KUKA KRL program: EPS_2_251825_SA28_A_20260116064107.src

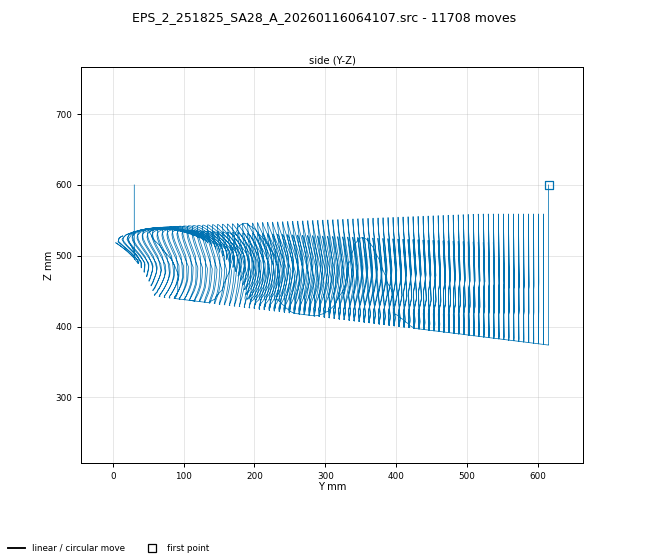
[picture p0: tool path of EPS_2_251825_SA28_A_20260116064107.src, 11708 of 11710 moves have a stored position in this frame; points joined in program order, loops and branches not executed]
&ACCESS RVP
&REL 4
&COMMENT QRS 19112012
&PARAM EDITMASK = *
DEF PART()
EXT BAS (BAS_COMMAND :IN,REAL :IN )
INT I
BAS (#INITMOV,0 )

;KUKA QRS Post kuka4.cps  Date:22-06-2017 !

File_ID=2987

QRS_PRE_INIT()

;Init var - Until changes are made in qrs_pre_init
Outlet_Square_prg=0
Inlet_1_Square_prg=0
Inlet_2_Square_prg=0
Inlet_3_Square_prg=0
Inlet_4_Square_prg=0
Inlet_5_Square_prg=0

Outlet_1={X 0.000, Y 520.860, Z 458.500, B 0.000, E1 0.000 }
Inlet_1={X 0.000, Y 523.760, Z 418.500, B 0.000, E1 223.000 }
Outlet_1_type=201
Inlet_1_type=201
;QRS#1=Sidecore dimensions
;QRS#2=200-8" PVC SDR 35
;QRS#3=200-8" PVC SDR 35
;QRS#4=
;QRS#5=
;QRS#6=
;QRS#7=
;QRS#8=
;QRS#9=12-08 PSX
;QRS#10=12-08 PSX
;QRS#11=
;QRS#12=
;QRS#13=
;QRS#14=
;QRS#15=
;QRS#16=1220x127x838 2,75'
;QRS#17=EPS Height
;QRS#18=559
;QRS#19=*
;QRS#20= UPDATED VERSION 22-06-2017
;QRS#21=*
Outlet_Square=0100
Inlet_1_Square=0100
Inlet_2_Square=0
Inlet_3_Square=0
Inlet_4_Square=0
Inlet_5_Square=0
Mill_Square=1
Outlet_Square_Prg=204
Inlet_1_Square_prg=204

QRS_INIT()

$ADVANCE=5

; T1
PTP {E1 173.612,E2 173.612}
PTP {X 0,Y 615.494,A -85,B 0,C 180,E1 173.612,E2 173.612,E3 0,E4 0,E5 0,E6 0}
QRS_SPEED_INIT()
LIN {X 0,Y 615.494,Z 600,A -85,B 0,C 180,E1 173.612,E2 173.612,E3 0,E4 0,E5 0,E6 0} C_VEL
LIN {X 0,Y 615.494,Z 383.874,A -85,B 0,C 180,E1 173.612,E2 173.612} C_VEL
LIN {X 0,Y 615.494,Z 375.697,A -85,B 0,C 180,E1 173.612,E2 173.612} C_VEL
LIN {X 0,Y 615.482,Z 373.697,A -85,B 0,C 180,E1 173.425,E2 173.425} C_VEL
LIN {X 0,Y 615.489,Z 373.696,A -85,B 0,C 180,E1 170.801,E2 170.801} C_VEL
LIN {X 0,Y 615.487,Z 373.7,A -85,B 0,C 180,E1 168.139,E2 168.139} C_VEL
LIN {X 0,Y 615.495,Z 373.697,A -85,B 0,C 180,E1 165.451,E2 165.451} C_VEL
LIN {X 0,Y 615.472,Z 373.699,A -85,B 0,C 180,E1 162.729,E2 162.729} C_VEL
LIN {X 0,Y 615.476,Z 373.7,A -85,B 0,C 180,E1 159.967,E2 159.967} C_VEL
LIN {X 0,Y 615.49,Z 373.699,A -85,B 0,C 180,E1 157.156,E2 157.156} C_VEL
LIN {X 0,Y 615.465,Z 373.701,A -85,B 0,C 180,E1 154.435,E2 154.435} C_VEL
LIN {X 0,Y 615.469,Z 373.7,A -85,B 0,C 180,E1 152.084,E2 152.084} C_VEL
LIN {X 0,Y 615.486,Z 373.698,A -85,B 0,C 180,E1 149.84,E2 149.84} C_VEL
LIN {X 0,Y 615.497,Z 373.697,A -85,B 0,C 180,E1 147.543,E2 147.543} C_VEL
LIN {X 0,Y 615.484,Z 373.7,A -85,B 0,C 180,E1 145.185,E2 145.185} C_VEL
LIN {X 0,Y 615.48,Z 373.7,A -85,B 0,C 180,E1 142.757,E2 142.757} C_VEL
LIN {X 0,Y 615.471,Z 373.699,A -85,B 0,C 180,E1 139.913,E2 139.913} C_VEL
LIN {X 0,Y 615.489,Z 373.701,A -85,B 0,C 180,E1 136.952,E2 136.952} C_VEL
LIN {X 0,Y 615.472,Z 373.699,A -85,B 0,C 180,E1 134.151,E2 134.151} C_VEL
LIN {X 0,Y 615.495,Z 373.694,A -85,B 0,C 180,E1 131.473,E2 131.473} C_VEL
LIN {X 0,Y 615.481,Z 373.7,A -85,B 0,C 180,E1 128.905,E2 128.905} C_VEL
LIN {X 0,Y 615.486,Z 373.7,A -85,B 0,C 180,E1 126.425,E2 126.425} C_VEL
LIN {X 0,Y 615.492,Z 373.696,A -85,B 0,C 180,E1 123.535,E2 123.535} C_VEL
LIN {X 0,Y 615.467,Z 373.7,A -85,B 0,C 180,E1 120.921,E2 120.921} C_VEL
LIN {X 0,Y 615.467,Z 373.7,A -85,B 0,C 180,E1 118.447,E2 118.447} C_VEL
LIN {X 0,Y 615.5,Z 373.699,A -85,B 0,C 180,E1 115.571,E2 115.571} C_VEL
LIN {X 0,Y 615.475,Z 373.7,A -85,B 0,C 180,E1 112.845,E2 112.845} C_VEL
LIN {X 0,Y 615.482,Z 373.697,A -85,B 0,C 180,E1 110.033,E2 110.033} C_VEL
LIN {X 0,Y 615.493,Z 373.7,A -85,B 0,C 180,E1 107.27,E2 107.27} C_VEL
LIN {X 0,Y 615.484,Z 373.699,A -85,B 0,C 180,E1 104.549,E2 104.549} C_VEL
LIN {X 0,Y 615.492,Z 373.694,A -85,B 0,C 180,E1 101.861,E2 101.861} C_VEL
LIN {X 0,Y 615.477,Z 373.699,A -85,B 0,C 180,E1 99.199,E2 99.199} C_VEL
LIN {X 0,Y 615.489,Z 373.7,A -85,B 0,C 180,E1 96.557,E2 96.557} C_VEL
LIN {X 0,Y 615.49,Z 373.699,A -85,B 0,C 180,E1 93.929,E2 93.929} C_VEL
LIN {X 0,Y 615.47,Z 373.7,A -85,B 0,C 180,E1 91.309,E2 91.309} C_VEL
LIN {X 0,Y 615.465,Z 373.7,A -85,B 0,C 180,E1 88.692,E2 88.692} C_VEL
LIN {X 0,Y 615.491,Z 373.696,A -85,B 0,C 180,E1 86.072,E2 86.072} C_VEL
LIN {X 0,Y 615.488,Z 373.701,A -85,B 0,C 180,E1 83.423,E2 83.423} C_VEL
LIN {X 0,Y 615.486,Z 373.972,A -85,B 0,C 180,E1 82.125,E2 82.125} C_VEL
LIN {X 0,Y 615.488,Z 378.125,A -85,B 0,C 180,E1 79.473,E2 79.473} C_VEL
LIN {X 0,Y 615.44,Z 382.418,A -85,B 0,C 180,E1 76.798,E2 76.798} C_VEL
LIN {X 0,Y 615.491,Z 386.897,A -85,B 0,C 180,E1 74.095,E2 74.095} C_VEL
LIN {X 0,Y 615.433,Z 391.562,A -85,B 0,C 180,E1 71.353,E2 71.353} C_VEL
LIN {X 0,Y 615.424,Z 395.176,A -85,B 0,C 180,E1 69.267,E2 69.267} C_VEL
LIN {X 0,Y 615.42,Z 398.895,A -85,B 0,C 180,E1 67.153,E2 67.153} C_VEL
LIN {X 0,Y 615.475,Z 403.743,A -85,B 0,C 180,E1 64.434,E2 64.434} C_VEL
LIN {X 0,Y 615.418,Z 408.949,A -85,B 0,C 180,E1 61.562,E2 61.562} C_VEL
LIN {X 0,Y 615.425,Z 413.511,A -85,B 0,C 180,E1 59.077,E2 59.077} C_VEL
LIN {X 0,Y 615.48,Z 414.447,A -85,B 0,C 180,E1 58.563,E2 58.563} C_VEL
LIN {X 0,Y 615.474,Z 430.159,A -85,B 0,C 180,E1 58.196,E2 58.196} C_VEL
LIN {X 0,Y 615.43,Z 442.777,A -85,B 0,C 180,E1 57.758,E2 57.758} C_VEL
LIN {X 0,Y 615.422,Z 453.783,A -85,B 0,C 180,E1 57.248,E2 57.248} C_VEL
LIN {X 0,Y 615.491,Z 465.713,A -85,B 0,C 180,E1 56.539,E2 56.539} C_VEL
LIN {X 0,Y 615.496,Z 475.546,A -85,B 0,C 180,E1 55.809,E2 55.809} C_VEL
LIN {X 0,Y 615.498,Z 484.561,A -85,B 0,C 180,E1 54.987,E2 54.987} C_VEL
LIN {X 0,Y 615.498,Z 493.211,A -85,B 0,C 180,E1 54.019,E2 54.019} C_VEL
LIN {X 0,Y 615.496,Z 500.126,A -85,B 0,C 180,E1 53.063,E2 53.063} C_VEL
LIN {X 0,Y 615.497,Z 506.555,A -85,B 0,C 180,E1 51.933,E2 51.933} C_VEL
LIN {X 0,Y 615.496,Z 510.941,A -85,B 0,C 180,E1 50.937,E2 50.937} C_VEL
LIN {X 0,Y 615.497,Z 514.331,A -85,B 0,C 180,E1 49.91,E2 49.91} C_VEL
LIN {X 0,Y 615.495,Z 516.63,A -85,B 0,C 180,E1 48.905,E2 48.905} C_VEL
LIN {X 0,Y 615.493,Z 518.147,A -85,B 0,C 180,E1 47.648,E2 47.648} C_VEL
LIN {X 0,Y 615.496,Z 518.347,A -85,B 0,C 180,E1 46.757,E2 46.757} C_VEL
LIN {X 0,Y 615.494,Z 517.823,A -85,B 0,C 180,E1 45.852,E2 45.852} C_VEL
LIN {X 0,Y 615.493,Z 516.511,A -85,B 0,C 180,E1 44.933,E2 44.933} C_VEL
LIN {X 0,Y 615.496,Z 513.199,A -85,B 0,C 180,E1 43.62,E2 43.62} C_VEL
LIN {X 0,Y 615.495,Z 508.364,A -85,B 0,C 180,E1 42.352,E2 42.352} C_VEL
LIN {X 0,Y 615.498,Z 502.814,A -85,B 0,C 180,E1 41.284,E2 41.284} C_VEL
LIN {X 0,Y 615.496,Z 496.693,A -85,B 0,C 180,E1 40.348,E2 40.348} C_VEL
LIN {X 0,Y 615.497,Z 489.1,A -85,B 0,C 180,E1 39.406,E2 39.406} C_VEL
LIN {X 0,Y 615.495,Z 479.987,A -85,B 0,C 180,E1 38.485,E2 38.485} C_VEL
LIN {X 0,Y 615.498,Z 470.716,A -85,B 0,C 180,E1 37.723,E2 37.723} C_VEL
LIN {X 0,Y 615.484,Z 460.045,A -85,B 0,C 180,E1 37.013,E2 37.013} C_VEL
LIN {X 0,Y 615.481,Z 448.967,A -85,B 0,C 180,E1 36.425,E2 36.425} C_VEL
LIN {X 0,Y 615.471,Z 437.295,A -85,B 0,C 180,E1 35.944,E2 35.944} C_VEL
LIN {X 0,Y 615.491,Z 424.587,A -85,B 0,C 180,E1 35.565,E2 35.565} C_VEL
LIN {X 0,Y 615.485,Z 414.432,A -85,B 0,C 180,E1 35.34,E2 35.34} C_VEL
LIN {X 0,Y 615.485,Z 409.134,A -85,B 0,C 180,E1 32.458,E2 32.458} C_VEL
LIN {X 0,Y 615.488,Z 404.309,A -85,B 0,C 180,E1 29.796,E2 29.796} C_VEL
LIN {X 0,Y 615.477,Z 399.396,A -85,B 0,C 180,E1 27.045,E2 27.045} C_VEL
LIN {X 0,Y 615.483,Z 394.517,A -85,B 0,C 180,E1 24.272,E2 24.272} C_VEL
LIN {X 0,Y 615.488,Z 390.83,A -85,B 0,C 180,E1 22.136,E2 22.136} C_VEL
LIN {X 0,Y 615.486,Z 387.261,A -85,B 0,C 180,E1 20.033,E2 20.033} C_VEL
LIN {X 0,Y 615.467,Z 382.675,A -85,B 0,C 180,E1 17.271,E2 17.271} C_VEL
LIN {X 0,Y 615.49,Z 378.323,A -85,B 0,C 180,E1 14.549,E2 14.549} C_VEL
LIN {X 0,Y 615.485,Z 374.113,A -85,B 0,C 180,E1 11.861,E2 11.861} C_VEL
LIN {X 0,Y 615.491,Z 373.699,A -85,B 0,C 180,E1 10.893,E2 10.893} C_VEL
LIN {X 0,Y 615.491,Z 373.7,A -85,B 0,C 180,E1 8.537,E2 8.537} C_VEL
LIN {X 0,Y 615.477,Z 373.7,A -85,B 0,C 180,E1 5.899,E2 5.899} C_VEL
LIN {X 0,Y 615.494,Z 373.698,A -85,B 0,C 180,E1 3.273,E2 3.273} C_VEL
LIN {X 0,Y 615.487,Z 373.698,A -85,B 0,C 180,E1 0.654,E2 0.654} C_VEL
LIN {X 0,Y 615.484,Z 373.7,A -85,B 0,C 180,E1 -1.963,E2 -1.963} C_VEL
LIN {X 0,Y 615.478,Z 373.7,A -85,B 0,C 180,E1 -4.585,E2 -4.585} C_VEL
LIN {X 0,Y 615.481,Z 373.7,A -85,B 0,C 180,E1 -7.216,E2 -7.216} C_VEL
LIN {X 0,Y 615.482,Z 373.7,A -85,B 0,C 180,E1 -9.862,E2 -9.862} C_VEL
LIN {X 0,Y 615.487,Z 373.698,A -85,B 0,C 180,E1 -12.53,E2 -12.53} C_VEL
LIN {X 0,Y 615.491,Z 373.701,A -85,B 0,C 180,E1 -15.226,E2 -15.226} C_VEL
LIN {X 0,Y 615.475,Z 373.7,A -85,B 0,C 180,E1 -17.957,E2 -17.957} C_VEL
LIN {X 0,Y 615.497,Z 373.697,A -85,B 0,C 180,E1 -20.73,E2 -20.73} C_VEL
LIN {X 0,Y 615.485,Z 373.702,A -85,B 0,C 180,E1 -23.557,E2 -23.557} C_VEL
LIN {X 0,Y 615.48,Z 373.7,A -85,B 0,C 180,E1 -26.445,E2 -26.445} C_VEL
LIN {X 0,Y 615.491,Z 373.699,A -85,B 0,C 180,E1 -28.658,E2 -28.658} C_VEL
LIN {X 0,Y 615.481,Z 373.701,A -85,B 0,C 180,E1 -31.086,E2 -31.086} C_VEL
LIN {X 0,Y 615.471,Z 373.701,A -85,B 0,C 180,E1 -33.533,E2 -33.533} C_VEL
LIN {X 0,Y 615.478,Z 373.701,A -85,B 0,C 180,E1 -35.833,E2 -35.833} C_VEL
LIN {X 0,Y 615.491,Z 373.7,A -85,B 0,C 180,E1 -38.068,E2 -38.068} C_VEL
LIN {X 0,Y 615.487,Z 373.699,A -85,B 0,C 180,E1 -41.095,E2 -41.095} C_VEL
LIN {X 0,Y 615.491,Z 373.699,A -85,B 0,C 180,E1 -43.245,E2 -43.245} C_VEL
LIN {X 0,Y 615.475,Z 373.7,A -85,B 0,C 180,E1 -46.004,E2 -46.004} C_VEL
LIN {X 0,Y 615.498,Z 373.7,A -85,B 0,C 180,E1 -48.528,E2 -48.528} C_VEL
LIN {X 0,Y 615.476,Z 373.7,A -85,B 0,C 180,E1 -51.095,E2 -51.095} C_VEL
LIN {X 0,Y 615.484,Z 373.7,A -85,B 0,C 180,E1 -53.576,E2 -53.576} C_VEL
LIN {X 0,Y 615.494,Z 373.898,A -85,B 0,C 180,E1 -54.586,E2 -54.586} C_VEL
LIN {X 0,Y 615.488,Z 381.521,A -85,B 0,C 180,E1 -57.155,E2 -57.155} C_VEL
LIN {X 0,Y 615.445,Z 389.797,A -85,B 0,C 180,E1 -59.838,E2 -59.838} C_VEL
LIN {X 0,Y 615.44,Z 399.232,A -85,B 0,C 180,E1 -62.821,E2 -62.821} C_VEL
LIN {X 0,Y 615.439,Z 406.311,A -85,B 0,C 180,E1 -65.007,E2 -65.007} C_VEL
LIN {X 0,Y 615.484,Z 415.038,A -85,B 0,C 180,E1 -67.655,E2 -67.655} C_VEL
LIN {X 0,Y 615.486,Z 423.98,A -85,B 0,C 180,E1 -70.315,E2 -70.315} C_VEL
LIN {X 0,Y 615.487,Z 433.396,A -85,B 0,C 180,E1 -73.072,E2 -73.072} C_VEL
LIN {X 0,Y 615.472,Z 442.71,A -85,B 0,C 180,E1 -75.759,E2 -75.759} C_VEL
LIN {X 0,Y 615.494,Z 451.992,A -85,B 0,C 180,E1 -78.369,E2 -78.369} C_VEL
LIN {X 0,Y 615.499,Z 464.077,A -85,B 0,C 180,E1 -78.599,E2 -78.599} C_VEL
LIN {X 0,Y 615.463,Z 476.74,A -85,B 0,C 180,E1 -78.968,E2 -78.968} C_VEL
LIN {X 0,Y 615.45,Z 489.035,A -85,B 0,C 180,E1 -79.473,E2 -79.473} C_VEL
LIN {X 0,Y 615.486,Z 499.987,A -85,B 0,C 180,E1 -80.055,E2 -80.055} C_VEL
LIN {X 0,Y 615.499,Z 511.172,A -85,B 0,C 180,E1 -80.802,E2 -80.802} C_VEL
LIN {X 0,Y 615.498,Z 521.048,A -85,B 0,C 180,E1 -81.629,E2 -81.629} C_VEL
LIN {X 0,Y 615.498,Z 530.609,A -85,B 0,C 180,E1 -82.62,E2 -82.62} C_VEL
LIN {X 0,Y 615.496,Z 538.205,A -85,B 0,C 180,E1 -83.608,E2 -83.608} C_VEL
LIN {X 0,Y 615.498,Z 545.206,A -85,B 0,C 180,E1 -84.759,E2 -84.759} C_VEL
LIN {X 0,Y 615.494,Z 549.852,A -85,B 0,C 180,E1 -85.744,E2 -85.744} C_VEL
LIN {X 0,Y 615.494,Z 553.4,A -85,B 0,C 180,E1 -86.727,E2 -86.727} C_VEL
LIN {X 0,Y 615.497,Z 555.234,A -85,B 0,C 180,E1 -87.382,E2 -87.382} C_VEL
LIN {X 0,Y 615.499,Z 556.608,A -85,B 0,C 180,E1 -88.037,E2 -88.037} C_VEL
LIN {X 0,Y 615.496,Z 558.174,A -85,B 0,C 180,E1 -89.346,E2 -89.346} C_VEL
LIN {X 0,Y 615.494,Z 558.389,A -85,B 0,C 180,E1 -90,E2 -90} C_VEL
LIN {X 0,Y 615.495,Z 557.58,A -85,B 0,C 180,E1 -91.309,E2 -91.309} C_VEL
LIN {X 0,Y 615.499,Z 556.607,A -85,B 0,C 180,E1 -91.963,E2 -91.963} C_VEL
LIN {X 0,Y 615.497,Z 555.232,A -85,B 0,C 180,E1 -92.618,E2 -92.618} C_VEL
LIN {X 0,Y 615.496,Z 552.349,A -85,B 0,C 180,E1 -93.601,E2 -93.601} C_VEL
LIN {X 0,Y 615.498,Z 548.44,A -85,B 0,C 180,E1 -94.585,E2 -94.585} C_VEL
LIN {X 0,Y 615.499,Z 543.404,A -85,B 0,C 180,E1 -95.57,E2 -95.57} C_VEL
LIN {X 0,Y 615.497,Z 536.87,A -85,B 0,C 180,E1 -96.583,E2 -96.583} C_VEL
LIN {X 0,Y 615.497,Z 529.131,A -85,B 0,C 180,E1 -97.546,E2 -97.546} C_VEL
LIN {X 0,Y 615.498,Z 521.043,A -85,B 0,C 180,E1 -98.371,E2 -98.371} C_VEL
LIN {X 0,Y 615.499,Z 511.165,A -85,B 0,C 180,E1 -99.199,E2 -99.199} C_VEL
LIN {X 0,Y 615.487,Z 499.978,A -85,B 0,C 180,E1 -99.945,E2 -99.945} C_VEL
LIN {X 0,Y 615.45,Z 489.025,A -85,B 0,C 180,E1 -100.528,E2 -100.528} C_VEL
LIN {X 0,Y 615.463,Z 476.734,A -85,B 0,C 180,E1 -101.032,E2 -101.032} C_VEL
LIN {X 0,Y 615.499,Z 464.055,A -85,B 0,C 180,E1 -101.402,E2 -101.402} C_VEL
LIN {X 0,Y 615.494,Z 451.773,A -85,B 0,C 180,E1 -101.652,E2 -101.652} C_VEL
LIN {X 0,Y 615.472,Z 442.709,A -85,B 0,C 180,E1 -104.241,E2 -104.241} C_VEL
LIN {X 0,Y 615.487,Z 433.394,A -85,B 0,C 180,E1 -106.928,E2 -106.928} C_VEL
LIN {X 0,Y 615.484,Z 423.979,A -85,B 0,C 180,E1 -109.685,E2 -109.685} C_VEL
LIN {X 0,Y 615.484,Z 415.038,A -85,B 0,C 180,E1 -112.344,E2 -112.344} C_VEL
LIN {X 0,Y 615.439,Z 406.31,A -85,B 0,C 180,E1 -114.994,E2 -114.994} C_VEL
LIN {X 0,Y 615.478,Z 398.047,A -85,B 0,C 180,E1 -117.546,E2 -117.546} C_VEL
LIN {X 0,Y 615.445,Z 389.795,A -85,B 0,C 180,E1 -120.162,E2 -120.162} C_VEL
LIN {X 0,Y 615.488,Z 381.521,A -85,B 0,C 180,E1 -122.846,E2 -122.846} C_VEL
LIN {X 0,Y 615.495,Z 373.695,A -85,B 0,C 180,E1 -125.515,E2 -125.515} C_VEL
LIN {X 0,Y 615.469,Z 373.7,A -85,B 0,C 180,E1 -128.07,E2 -128.07} C_VEL
LIN {X 0,Y 615.467,Z 373.7,A -85,B 0,C 180,E1 -130.608,E2 -130.608} C_VEL
LIN {X 0,Y 615.477,Z 373.7,A -85,B 0,C 180,E1 -133.246,E2 -133.246} C_VEL
LIN {X 0,Y 615.488,Z 373.7,A -85,B 0,C 180,E1 -136.002,E2 -136.002} C_VEL
LIN {X 0,Y 615.478,Z 373.7,A -85,B 0,C 180,E1 -138.525,E2 -138.525} C_VEL
LIN {X 0,Y 615.485,Z 373.697,A -85,B 0,C 180,E1 -141.095,E2 -141.095} C_VEL
LIN {X 0,Y 615.484,Z 373.696,A -85,B 0,C 180,E1 -143.575,E2 -143.575} C_VEL
LIN {X 0,Y 615.481,Z 373.701,A -85,B 0,C 180,E1 -146.467,E2 -146.467} C_VEL
LIN {X 0,Y 615.492,Z 373.701,A -85,B 0,C 180,E1 -149.08,E2 -149.08} C_VEL
LIN {X 0,Y 615.485,Z 373.7,A -85,B 0,C 180,E1 -151.55,E2 -151.55} C_VEL
LIN {X 0,Y 615.468,Z 373.7,A -85,B 0,C 180,E1 -154.283,E2 -154.283} C_VEL
LIN {X 0,Y 615.491,Z 373.698,A -85,B 0,C 180,E1 -157.155,E2 -157.155} C_VEL
LIN {X 0,Y 615.482,Z 373.7,A -85,B 0,C 180,E1 -159.967,E2 -159.967} C_VEL
LIN {X 0,Y 615.475,Z 373.698,A -85,B 0,C 180,E1 -162.729,E2 -162.729} C_VEL
LIN {X 0,Y 615.493,Z 373.696,A -85,B 0,C 180,E1 -165.451,E2 -165.451} C_VEL
LIN {X 0,Y 615.487,Z 373.702,A -85,B 0,C 180,E1 -168.139,E2 -168.139} C_VEL
LIN {X 0,Y 615.492,Z 373.696,A -85,B 0,C 180,E1 -170.801,E2 -170.801} C_VEL
LIN {X 0,Y 615.477,Z 373.698,A -85,B 0,C 180,E1 -173.443,E2 -173.443} C_VEL
LIN {X 0,Y 615.471,Z 373.7,A -85,B 0,C 180,E1 -176.071,E2 -176.071} C_VEL
LIN {X 0,Y 615.483,Z 373.7,A -85,B 0,C 180,E1 -178.691,E2 -178.691} C_VEL
LIN {X 0,Y 615.489,Z 373.701,A -85,B 0,C 180,E1 -181.309,E2 -181.309} C_VEL
LIN {X 0,Y 615.475,Z 373.7,A -85,B 0,C 180,E1 -183.929,E2 -183.929} C_VEL
LIN {X 0,Y 615.482,Z 373.697,A -85,B 0,C 180,E1 -186.575,E2 -186.575} C_VEL
LIN {X 0,Y 614.812,Z 373.846,A -85,B 0,C 180,E1 -187.121,E2 -187.121} C_VEL
LIN {X 0,Y 611.983,Z 374.255,A -85,B 0,C 180,E1 -188.007,E2 -188.007} C_VEL
LIN {X 0,Y 609.591,Z 374.565,A -85,B 0,C 180,E1 -188.719,E2 -188.719} C_VEL
LIN {X 0,Y 608.55,Z 374.684,A -85,B 0,C 180,E1 -189.269,E2 -189.269} C_VEL
LIN {X 0,Y 608.458,Z 374.694,A -85,B 0,C 180,E1 -189.455,E2 -189.455} C_VEL
LIN {X 0,Y 608.461,Z 374.697,A -85,B 0,C 180,E1 -192,E2 -192} C_VEL
LIN {X 0,Y 608.481,Z 374.692,A -85,B 0,C 180,E1 -194.72,E2 -194.72} C_VEL
LIN {X 0,Y 608.447,Z 374.695,A -85,B 0,C 180,E1 -197.477,E2 -197.477} C_VEL
LIN {X 0,Y 608.461,Z 374.697,A -85,B 0,C 180,E1 -200.274,E2 -200.274} C_VEL
LIN {X 0,Y 608.448,Z 374.695,A -85,B 0,C 180,E1 -203.124,E2 -203.124} C_VEL
LIN {X 0,Y 608.454,Z 374.694,A -85,B 0,C 180,E1 -205.718,E2 -205.718} C_VEL
LIN {X 0,Y 608.441,Z 374.696,A -85,B 0,C 180,E1 -208.267,E2 -208.267} C_VEL
LIN {X 0,Y 608.474,Z 374.692,A -85,B 0,C 180,E1 -210.545,E2 -210.545} C_VEL
LIN {X 0,Y 608.463,Z 374.693,A -85,B 0,C 180,E1 -212.879,E2 -212.879} C_VEL
LIN {X 0,Y 608.438,Z 374.696,A -85,B 0,C 180,E1 -215.278,E2 -215.278} C_VEL
LIN {X 0,Y 608.465,Z 374.693,A -85,B 0,C 180,E1 -217.747,E2 -217.747} C_VEL
LIN {X 0,Y 608.444,Z 374.697,A -85,B 0,C 180,E1 -220.328,E2 -220.328} C_VEL
LIN {X 0,Y 608.455,Z 374.698,A -85,B 0,C 180,E1 -222.96,E2 -222.96} C_VEL
LIN {X 0,Y 608.444,Z 374.696,A -85,B 0,C 180,E1 -225.737,E2 -225.737} C_VEL
LIN {X 0,Y 608.469,Z 374.693,A -85,B 0,C 180,E1 -228.657,E2 -228.657} C_VEL
LIN {X 0,Y 608.458,Z 374.694,A -85,B 0,C 180,E1 -231.761,E2 -231.761} C_VEL
LIN {X 0,Y 608.48,Z 374.693,A -85,B 0,C 180,E1 -233.95,E2 -233.95} C_VEL
LIN {X 0,Y 608.467,Z 374.694,A -85,B 0,C 180,E1 -236.329,E2 -236.329} C_VEL
LIN {X 0,Y 608.444,Z 374.697,A -85,B 0,C 180,E1 -238.733,E2 -238.733} C_VEL
LIN {X 0,Y 608.458,Z 374.694,A -85,B 0,C 180,E1 -241.383,E2 -241.383} C_VEL
LIN {X 0,Y 608.483,Z 374.693,A -85,B 0,C 180,E1 -244.277,E2 -244.277} C_VEL
LIN {X 0,Y 608.448,Z 374.699,A -85,B 0,C 180,E1 -246.876,E2 -246.876} C_VEL
LIN {X 0,Y 608.458,Z 374.694,A -85,B 0,C 180,E1 -249.726,E2 -249.726} C_VEL
LIN {X 0,Y 608.459,Z 374.695,A -85,B 0,C 180,E1 -252.524,E2 -252.524} C_VEL
LIN {X 0,Y 608.471,Z 374.695,A -85,B 0,C 180,E1 -255.279,E2 -255.279} C_VEL
LIN {X 0,Y 608.465,Z 374.693,A -85,B 0,C 180,E1 -258,E2 -258} C_VEL
LIN {X 0,Y 608.464,Z 374.693,A -85,B 0,C 180,E1 -260.694,E2 -260.694} C_VEL
LIN {X 0,Y 608.482,Z 374.693,A -85,B 0,C 180,E1 -263.367,E2 -263.367} C_VEL
LIN {X 0,Y 608.457,Z 374.697,A -85,B 0,C 180,E1 -266.026,E2 -266.026} C_VEL
LIN {X 0,Y 608.457,Z 374.695,A -85,B 0,C 180,E1 -268.676,E2 -268.676} C_VEL
LIN {X 0,Y 608.452,Z 374.694,A -85,B 0,C 180,E1 -271.323,E2 -271.323} C_VEL
LIN {X 0,Y 608.459,Z 374.695,A -85,B 0,C 180,E1 -273.974,E2 -273.974} C_VEL
LIN {X 0,Y 608.481,Z 374.694,A -85,B 0,C 180,E1 -276.632,E2 -276.632} C_VEL
LIN {X 0,Y 608.445,Z 375.038,A -85,B 0,C 180,E1 -277.967,E2 -277.967} C_VEL
LIN {X 0,Y 608.445,Z 379.215,A -85,B 0,C 180,E1 -280.65,E2 -280.65} C_VEL
LIN {X 0,Y 608.422,Z 382.419,A -85,B 0,C 180,E1 -282.678,E2 -282.678} C_VEL
LIN {X 0,Y 608.41,Z 385.764,A -85,B 0,C 180,E1 -284.722,E2 -284.722} C_VEL
LIN {X 0,Y 608.383,Z 389.208,A -85,B 0,C 180,E1 -286.786,E2 -286.786} C_VEL
LIN {X 0,Y 608.372,Z 392.751,A -85,B 0,C 180,E1 -288.872,E2 -288.872} C_VEL
LIN {X 0,Y 608.367,Z 396.398,A -85,B 0,C 180,E1 -290.984,E2 -290.984} C_VEL
LIN {X 0,Y 608.416,Z 401.421,A -85,B 0,C 180,E1 -293.847,E2 -293.847} C_VEL
LIN {X 0,Y 608.398,Z 405.33,A -85,B 0,C 180,E1 -296.037,E2 -296.037} C_VEL
LIN {X 0,Y 608.35,Z 409.959,A -85,B 0,C 180,E1 -298.598,E2 -298.598} C_VEL
LIN {X 0,Y 608.364,Z 413.52,A -85,B 0,C 180,E1 -300.55,E2 -300.55} C_VEL
LIN {X 0,Y 608.411,Z 414.959,A -85,B 0,C 180,E1 -301.319,E2 -301.319} C_VEL
LIN {X 0,Y 608.52,Z 427.755,A -85,B 0,C 180,E1 -301.604,E2 -301.604} C_VEL
LIN {X 0,Y 608.481,Z 441.098,A -85,B 0,C 180,E1 -302.044,E2 -302.044} C_VEL
LIN {X 0,Y 608.431,Z 452.961,A -85,B 0,C 180,E1 -302.58,E2 -302.58} C_VEL
LIN {X 0,Y 608.467,Z 464.767,A -85,B 0,C 180,E1 -303.273,E2 -303.273} C_VEL
LIN {X 0,Y 608.471,Z 475.592,A -85,B 0,C 180,E1 -304.07,E2 -304.07} C_VEL
LIN {X 0,Y 608.456,Z 484.744,A -85,B 0,C 180,E1 -304.906,E2 -304.906} C_VEL
LIN {X 0,Y 608.447,Z 493.214,A -85,B 0,C 180,E1 -305.854,E2 -305.854} C_VEL
LIN {X 0,Y 608.437,Z 500.875,A -85,B 0,C 180,E1 -306.916,E2 -306.916} C_VEL
LIN {X 0,Y 608.452,Z 506.951,A -85,B 0,C 180,E1 -307.99,E2 -307.99} C_VEL
LIN {X 0,Y 608.438,Z 511.188,A -85,B 0,C 180,E1 -308.94,E2 -308.94} C_VEL
LIN {X 0,Y 608.438,Z 514.392,A -85,B 0,C 180,E1 -309.871,E2 -309.871} C_VEL
LIN {X 0,Y 608.431,Z 517.399,A -85,B 0,C 180,E1 -311.178,E2 -311.178} C_VEL
LIN {X 0,Y 608.435,Z 518.747,A -85,B 0,C 180,E1 -312.331,E2 -312.331} C_VEL
LIN {X 0,Y 608.432,Z 518.945,A -85,B 0,C 180,E1 -313.305,E2 -313.305} C_VEL
LIN {X 0,Y 608.417,Z 518.312,A -85,B 0,C 180,E1 -314.26,E2 -314.26} C_VEL
LIN {X 0,Y 608.418,Z 516.889,A -85,B 0,C 180,E1 -315.2,E2 -315.2} C_VEL
LIN {X 0,Y 608.429,Z 514.653,A -85,B 0,C 180,E1 -316.127,E2 -316.127} C_VEL
LIN {X 0,Y 608.437,Z 511.603,A -85,B 0,C 180,E1 -317.039,E2 -317.039} C_VEL
LIN {X 0,Y 608.432,Z 507.748,A -85,B 0,C 180,E1 -317.936,E2 -317.936} C_VEL
LIN {X 0,Y 608.442,Z 501.685,A -85,B 0,C 180,E1 -319.042,E2 -319.042} C_VEL
LIN {X 0,Y 608.465,Z 494.077,A -85,B 0,C 180,E1 -320.13,E2 -320.13} C_VEL
LIN {X 0,Y 608.453,Z 485.632,A -85,B 0,C 180,E1 -321.093,E2 -321.093} C_VEL
LIN {X 0,Y 608.485,Z 475.757,A -85,B 0,C 180,E1 -322.006,E2 -322.006} C_VEL
LIN {X 0,Y 608.495,Z 465.897,A -85,B 0,C 180,E1 -322.742,E2 -322.742} C_VEL
LIN {X 0,Y 608.51,Z 455.007,A -85,B 0,C 180,E1 -323.399,E2 -323.399} C_VEL
LIN {X 0,Y 608.492,Z 443.492,A -85,B 0,C 180,E1 -323.948,E2 -323.948} C_VEL
LIN {X 0,Y 608.536,Z 431.712,A -85,B 0,C 180,E1 -324.373,E2 -324.373} C_VEL
LIN {X 0,Y 608.535,Z 418.492,A -85,B 0,C 180,E1 -324.703,E2 -324.703} C_VEL
LIN {X 0,Y 608.445,Z 414.919,A -85,B 0,C 180,E1 -324.776,E2 -324.776} C_VEL
LIN {X 0,Y 608.417,Z 409.971,A -85,B 0,C 180,E1 -327.483,E2 -327.483} C_VEL
LIN {X 0,Y 608.437,Z 405.03,A -85,B 0,C 180,E1 -330.219,E2 -330.219} C_VEL
LIN {X 0,Y 608.418,Z 400.432,A -85,B 0,C 180,E1 -332.802,E2 -332.802} C_VEL
LIN {X 0,Y 608.418,Z 395.835,A -85,B 0,C 180,E1 -335.427,E2 -335.427} C_VEL
LIN {X 0,Y 608.435,Z 390.89,A -85,B 0,C 180,E1 -338.307,E2 -338.307} C_VEL
LIN {X 0,Y 608.421,Z 387.323,A -85,B 0,C 180,E1 -340.428,E2 -340.428} C_VEL
LIN {X 0,Y 608.442,Z 382.736,A -85,B 0,C 180,E1 -343.216,E2 -343.216} C_VEL
LIN {X 0,Y 608.471,Z 378.395,A -85,B 0,C 180,E1 -345.98,E2 -345.98} C_VEL
LIN {X 0,Y 608.459,Z 375.259,A -85,B 0,C 180,E1 -348,E2 -348} C_VEL
LIN {X 0,Y 608.469,Z 374.694,A -85,B 0,C 180,E1 -349.041,E2 -349.041} C_VEL
LIN {X 0,Y 608.46,Z 374.698,A -85,B 0,C 180,E1 -351.364,E2 -351.364} C_VEL
LIN {X 0,Y 608.452,Z 374.695,A -85,B 0,C 180,E1 -354.033,E2 -354.033} C_VEL
LIN {X 0,Y 608.485,Z 374.693,A -85,B 0,C 180,E1 -356.689,E2 -356.689} C_VEL
LIN {X 0,Y 608.481,Z 374.692,A -85,B 0,C 180,E1 -359.338,E2 -359.338} C_VEL
LIN {X 0,Y 608.454,Z 374.696,A -85,B 0,C 180,E1 -361.986,E2 -361.986} C_VEL
LIN {X 0,Y 608.447,Z 374.697,A -85,B 0,C 180,E1 -364.638,E2 -364.638} C_VEL
LIN {X 0,Y 608.46,Z 374.695,A -85,B 0,C 180,E1 -367.3,E2 -367.3} C_VEL
LIN {X 0,Y 608.453,Z 374.697,A -85,B 0,C 180,E1 -369.977,E2 -369.977} C_VEL
LIN {X 0,Y 608.478,Z 374.692,A -85,B 0,C 180,E1 -372.677,E2 -372.677} C_VEL
LIN {X 0,Y 608.471,Z 374.695,A -85,B 0,C 180,E1 -375.406,E2 -375.406} C_VEL
LIN {X 0,Y 608.444,Z 374.697,A -85,B 0,C 180,E1 -378.172,E2 -378.172} C_VEL
LIN {X 0,Y 608.463,Z 374.694,A -85,B 0,C 180,E1 -380.981,E2 -380.981} C_VEL
LIN {X 0,Y 608.454,Z 374.695,A -85,B 0,C 180,E1 -383.124,E2 -383.124} C_VEL
LIN {X 0,Y 608.448,Z 374.696,A -85,B 0,C 180,E1 -386.036,E2 -386.036} C_VEL
LIN {X 0,Y 608.473,Z 374.694,A -85,B 0,C 180,E1 -388.621,E2 -388.621} C_VEL
LIN {X 0,Y 608.456,Z 374.695,A -85,B 0,C 180,E1 -391.317,E2 -391.317} C_VEL
LIN {X 0,Y 608.468,Z 374.694,A -85,B 0,C 180,E1 -393.735,E2 -393.735} C_VEL
LIN {X 0,Y 608.474,Z 374.696,A -85,B 0,C 180,E1 -396.091,E2 -396.091} C_VEL
LIN {X 0,Y 608.472,Z 374.693,A -85,B 0,C 180,E1 -398.588,E2 -398.588} C_VEL
LIN {X 0,Y 608.462,Z 374.697,A -85,B 0,C 180,E1 -401.343,E2 -401.343} C_VEL
LIN {X 0,Y 608.449,Z 374.697,A -85,B 0,C 180,E1 -404.264,E2 -404.264} C_VEL
LIN {X 0,Y 608.443,Z 374.696,A -85,B 0,C 180,E1 -407.04,E2 -407.04} C_VEL
LIN {X 0,Y 608.451,Z 374.698,A -85,B 0,C 180,E1 -409.697,E2 -409.697} C_VEL
LIN {X 0,Y 608.473,Z 374.693,A -85,B 0,C 180,E1 -412.255,E2 -412.255} C_VEL
LIN {X 0,Y 608.501,Z 374.786,A -85,B 0,C 180,E1 -414.422,E2 -414.422} C_VEL
LIN {X 0,Y 608.496,Z 382.695,A -85,B 0,C 180,E1 -417.123,E2 -417.123} C_VEL
LIN {X 0,Y 608.436,Z 389.845,A -85,B 0,C 180,E1 -419.454,E2 -419.454} C_VEL
LIN {X 0,Y 608.43,Z 396.945,A -85,B 0,C 180,E1 -421.733,E2 -421.733} C_VEL
LIN {X 0,Y 608.496,Z 405.034,A -85,B 0,C 180,E1 -424.275,E2 -424.275} C_VEL
LIN {X 0,Y 608.431,Z 413.511,A -85,B 0,C 180,E1 -426.876,E2 -426.876} C_VEL
LIN {X 0,Y 608.467,Z 421.624,A -85,B 0,C 180,E1 -429.322,E2 -429.322} C_VEL
LIN {X 0,Y 608.447,Z 431.261,A -85,B 0,C 180,E1 -432.176,E2 -432.176} C_VEL
LIN {X 0,Y 608.434,Z 440.728,A -85,B 0,C 180,E1 -434.936,E2 -434.936} C_VEL
LIN {X 0,Y 608.429,Z 450.195,A -85,B 0,C 180,E1 -437.661,E2 -437.661} C_VEL
LIN {X 0,Y 608.439,Z 452.192,A -85,B 0,C 180,E1 -438.233,E2 -438.233} C_VEL
LIN {X 0,Y 608.548,Z 465.109,A -85,B 0,C 180,E1 -438.488,E2 -438.488} C_VEL
LIN {X 0,Y 608.49,Z 477.491,A -85,B 0,C 180,E1 -438.864,E2 -438.864} C_VEL
LIN {X 0,Y 608.474,Z 489.179,A -85,B 0,C 180,E1 -439.351,E2 -439.351} C_VEL
LIN {X 0,Y 608.486,Z 501.584,A -85,B 0,C 180,E1 -440.024,E2 -440.024} C_VEL
LIN {X 0,Y 608.483,Z 512.478,A -85,B 0,C 180,E1 -440.779,E2 -440.779} C_VEL
LIN {X 0,Y 608.475,Z 523.115,A -85,B 0,C 180,E1 -441.699,E2 -441.699} C_VEL
LIN {X 0,Y 608.471,Z 530.963,A -85,B 0,C 180,E1 -442.534,E2 -442.534} C_VEL
LIN {X 0,Y 608.46,Z 538.288,A -85,B 0,C 180,E1 -443.485,E2 -443.485} C_VEL
LIN {X 0,Y 608.45,Z 543.867,A -85,B 0,C 180,E1 -444.366,E2 -444.366} C_VEL
LIN {X 0,Y 608.432,Z 548.951,A -85,B 0,C 180,E1 -445.362,E2 -445.362} C_VEL
LIN {X 0,Y 608.449,Z 552.897,A -85,B 0,C 180,E1 -446.358,E2 -446.358} C_VEL
LIN {X 0,Y 608.425,Z 555.81,A -85,B 0,C 180,E1 -447.352,E2 -447.352} C_VEL
LIN {X 0,Y 608.444,Z 557.202,A -85,B 0,C 180,E1 -448.014,E2 -448.014} C_VEL
LIN {X 0,Y 608.438,Z 558.784,A -85,B 0,C 180,E1 -449.338,E2 -449.338} C_VEL
LIN {X 0,Y 608.434,Z 559,A -85,B 0,C 180,E1 -450,E2 -450} C_VEL
LIN {X 0,Y 608.448,Z 558.183,A -85,B 0,C 180,E1 -451.324,E2 -451.324} C_VEL
LIN {X 0,Y 608.444,Z 557.201,A -85,B 0,C 180,E1 -451.986,E2 -451.986} C_VEL
LIN {X 0,Y 608.425,Z 555.809,A -85,B 0,C 180,E1 -452.648,E2 -452.648} C_VEL
LIN {X 0,Y 608.449,Z 552.895,A -85,B 0,C 180,E1 -453.643,E2 -453.643} C_VEL
LIN {X 0,Y 608.432,Z 548.949,A -85,B 0,C 180,E1 -454.638,E2 -454.638} C_VEL
LIN {X 0,Y 608.437,Z 542.875,A -85,B 0,C 180,E1 -455.801,E2 -455.801} C_VEL
LIN {X 0,Y 608.462,Z 536.233,A -85,B 0,C 180,E1 -456.8,E2 -456.8} C_VEL
LIN {X 0,Y 608.456,Z 527.987,A -85,B 0,C 180,E1 -457.8,E2 -457.8} C_VEL
LIN {X 0,Y 608.472,Z 519.534,A -85,B 0,C 180,E1 -458.636,E2 -458.636} C_VEL
LIN {X 0,Y 608.481,Z 509.088,A -85,B 0,C 180,E1 -459.474,E2 -459.474} C_VEL
LIN {X 0,Y 608.499,Z 498.753,A -85,B 0,C 180,E1 -460.145,E2 -460.145} C_VEL
LIN {X 0,Y 608.473,Z 487.82,A -85,B 0,C 180,E1 -460.715,E2 -460.715} C_VEL
LIN {X 0,Y 608.495,Z 476.059,A -85,B 0,C 180,E1 -461.187,E2 -461.187} C_VEL
LIN {X 0,Y 608.549,Z 463.259,A -85,B 0,C 180,E1 -461.555,E2 -461.555} C_VEL
LIN {X 0,Y 608.439,Z 452.19,A -85,B 0,C 180,E1 -461.768,E2 -461.768} C_VEL
LIN {X 0,Y 608.418,Z 443.093,A -85,B 0,C 180,E1 -464.38,E2 -464.38} C_VEL
LIN {X 0,Y 608.451,Z 434.81,A -85,B 0,C 180,E1 -466.784,E2 -466.784} C_VEL
LIN {X 0,Y 608.453,Z 425.343,A -85,B 0,C 180,E1 -469.571,E2 -469.571} C_VEL
LIN {X 0,Y 608.462,Z 415.643,A -85,B 0,C 180,E1 -472.476,E2 -472.476} C_VEL
LIN {X 0,Y 608.429,Z 407.593,A -85,B 0,C 180,E1 -474.937,E2 -474.937} C_VEL
LIN {X 0,Y 608.46,Z 399.31,A -85,B 0,C 180,E1 -477.518,E2 -477.518} C_VEL
LIN {X 0,Y 608.472,Z 391.613,A -85,B 0,C 180,E1 -479.972,E2 -479.972} C_VEL
LIN {X 0,Y 608.489,Z 383.769,A -85,B 0,C 180,E1 -482.526,E2 -482.526} C_VEL
LIN {X 0,Y 608.524,Z 375.662,A -85,B 0,C 180,E1 -485.272,E2 -485.272} C_VEL
LIN {X 0,Y 608.485,Z 374.691,A -85,B 0,C 180,E1 -485.681,E2 -485.681} C_VEL
LIN {X 0,Y 608.437,Z 374.699,A -85,B 0,C 180,E1 -488.59,E2 -488.59} C_VEL
LIN {X 0,Y 608.466,Z 374.694,A -85,B 0,C 180,E1 -491.342,E2 -491.342} C_VEL
LIN {X 0,Y 608.441,Z 374.696,A -85,B 0,C 180,E1 -494.262,E2 -494.262} C_VEL
LIN {X 0,Y 608.453,Z 374.698,A -85,B 0,C 180,E1 -497.04,E2 -497.04} C_VEL
LIN {X 0,Y 608.453,Z 374.696,A -85,B 0,C 180,E1 -499.697,E2 -499.697} C_VEL
LIN {X 0,Y 608.466,Z 374.693,A -85,B 0,C 180,E1 -502.253,E2 -502.253} C_VEL
LIN {X 0,Y 608.446,Z 374.696,A -85,B 0,C 180,E1 -505.095,E2 -505.095} C_VEL
LIN {X 0,Y 608.467,Z 374.696,A -85,B 0,C 180,E1 -507.905,E2 -507.905} C_VEL
LIN {X 0,Y 608.48,Z 374.695,A -85,B 0,C 180,E1 -510.221,E2 -510.221} C_VEL
LIN {X 0,Y 608.482,Z 374.693,A -85,B 0,C 180,E1 -512.792,E2 -512.792} C_VEL
LIN {X 0,Y 608.476,Z 374.692,A -85,B 0,C 180,E1 -515.848,E2 -515.848} C_VEL
LIN {X 0,Y 608.469,Z 374.694,A -85,B 0,C 180,E1 -518.308,E2 -518.308} C_VEL
LIN {X 0,Y 608.471,Z 374.693,A -85,B 0,C 180,E1 -521.283,E2 -521.283} C_VEL
LIN {X 0,Y 608.448,Z 374.695,A -85,B 0,C 180,E1 -523.906,E2 -523.906} C_VEL
LIN {X 0,Y 608.46,Z 374.695,A -85,B 0,C 180,E1 -526.643,E2 -526.643} C_VEL
LIN {X 0,Y 608.464,Z 374.696,A -85,B 0,C 180,E1 -529.35,E2 -529.35} C_VEL
LIN {X 0,Y 608.465,Z 374.694,A -85,B 0,C 180,E1 -532.033,E2 -532.033} C_VEL
LIN {X 0,Y 608.462,Z 374.693,A -85,B 0,C 180,E1 -534.698,E2 -534.698} C_VEL
LIN {X 0,Y 608.482,Z 374.692,A -85,B 0,C 180,E1 -537.352,E2 -537.352} C_VEL
LIN {X 0,Y 608.477,Z 374.695,A -85,B 0,C 180,E1 -540,E2 -540} C_VEL
LIN {X 0,Y 608.484,Z 374.692,A -85,B 0,C 180,E1 -542.648,E2 -542.648} C_VEL
LIN {X 0,Y 608.46,Z 374.694,A -85,B 0,C 180,E1 -545.302,E2 -545.302} C_VEL
LIN {X 0,Y 608.465,Z 374.693,A -85,B 0,C 180,E1 -547.967,E2 -547.967} C_VEL
LIN {X 0,Y 608.458,Z 374.694,A -85,B 0,C 180,E1 -549.455,E2 -549.455} C_VEL
LIN {X 0,Y 607.774,Z 374.78,A -85,B 0,C 180,E1 -550.008,E2 -550.008} C_VEL
LIN {X 0,Y 604.92,Z 375.137,A -85,B 0,C 180,E1 -550.905,E2 -550.905} C_VEL
LIN {X 0,Y 602.521,Z 375.436,A -85,B 0,C 180,E1 -551.626,E2 -551.626} C_VEL
LIN {X 0,Y 601.492,Z 375.564,A -85,B 0,C 180,E1 -552.183,E2 -552.183} C_VEL
LIN {X 0,Y 601.408,Z 375.572,A -85,B 0,C 180,E1 -552.371,E2 -552.371} C_VEL
LIN {X 0,Y 601.433,Z 375.569,A -85,B 0,C 180,E1 -554.897,E2 -554.897} C_VEL
LIN {X 0,Y 601.395,Z 375.575,A -85,B 0,C 180,E1 -557.688,E2 -557.688} C_VEL
LIN {X 0,Y 601.435,Z 375.57,A -85,B 0,C 180,E1 -560.522,E2 -560.522} C_VEL
LIN {X 0,Y 601.419,Z 375.571,A -85,B 0,C 180,E1 -563.41,E2 -563.41} C_VEL
LIN {X 0,Y 601.401,Z 375.576,A -85,B 0,C 180,E1 -566.364,E2 -566.364} C_VEL
LIN {X 0,Y 601.427,Z 375.572,A -85,B 0,C 180,E1 -568.787,E2 -568.787} C_VEL
LIN {X 0,Y 601.419,Z 375.571,A -85,B 0,C 180,E1 -571.455,E2 -571.455} C_VEL
LIN {X 0,Y 601.428,Z 375.569,A -85,B 0,C 180,E1 -574.118,E2 -574.118} C_VEL
LIN {X 0,Y 601.419,Z 375.571,A -85,B 0,C 180,E1 -576.582,E2 -576.582} C_VEL
LIN {X 0,Y 601.411,Z 375.573,A -85,B 0,C 180,E1 -579.127,E2 -579.127} C_VEL
LIN {X 0,Y 601.422,Z 375.574,A -85,B 0,C 180,E1 -581.765,E2 -581.765} C_VEL
LIN {X 0,Y 601.426,Z 375.57,A -85,B 0,C 180,E1 -584.535,E2 -584.535} C_VEL
LIN {X 0,Y 601.411,Z 375.572,A -85,B 0,C 180,E1 -587.41,E2 -587.41} C_VEL
LIN {X 0,Y 601.404,Z 375.575,A -85,B 0,C 180,E1 -590.004,E2 -590.004} C_VEL
LIN {X 0,Y 601.434,Z 375.572,A -85,B 0,C 180,E1 -592.618,E2 -592.618} C_VEL
LIN {X 0,Y 601.404,Z 375.574,A -85,B 0,C 180,E1 -595.067,E2 -595.067} C_VEL
LIN {X 0,Y 601.428,Z 375.571,A -85,B 0,C 180,E1 -597.484,E2 -597.484} C_VEL
LIN {X 0,Y 601.431,Z 375.571,A -85,B 0,C 180,E1 -599.851,E2 -599.851} C_VEL
LIN {X 0,Y 601.447,Z 375.568,A -85,B 0,C 180,E1 -602.889,E2 -602.889} C_VEL
LIN {X 0,Y 601.46,Z 375.567,A -85,B 0,C 180,E1 -605.86,E2 -605.86} C_VEL
LIN {X 0,Y 601.406,Z 375.572,A -85,B 0,C 180,E1 -608.761,E2 -608.761} C_VEL
LIN {X 0,Y 601.422,Z 375.574,A -85,B 0,C 180,E1 -611.608,E2 -611.608} C_VEL
LIN {X 0,Y 601.41,Z 375.572,A -85,B 0,C 180,E1 -614.408,E2 -614.408} C_VEL
LIN {X 0,Y 601.415,Z 375.571,A -85,B 0,C 180,E1 -617.172,E2 -617.172} C_VEL
LIN {X 0,Y 601.434,Z 375.572,A -85,B 0,C 180,E1 -619.905,E2 -619.905} C_VEL
LIN {X 0,Y 601.408,Z 375.573,A -85,B 0,C 180,E1 -622.614,E2 -622.614} C_VEL
LIN {X 0,Y 601.408,Z 375.572,A -85,B 0,C 180,E1 -625.308,E2 -625.308} C_VEL
LIN {X 0,Y 601.437,Z 375.569,A -85,B 0,C 180,E1 -627.991,E2 -627.991} C_VEL
LIN {X 0,Y 601.455,Z 375.57,A -85,B 0,C 180,E1 -630.669,E2 -630.669} C_VEL
LIN {X 0,Y 601.433,Z 375.57,A -85,B 0,C 180,E1 -633.349,E2 -633.349} C_VEL
LIN {X 0,Y 601.423,Z 375.57,A -85,B 0,C 180,E1 -636.037,E2 -636.037} C_VEL
LIN {X 0,Y 601.386,Z 375.575,A -85,B 0,C 180,E1 -637.385,E2 -637.385} C_VEL
LIN {X 0,Y 601.388,Z 375.929,A -85,B 0,C 180,E1 -638.061,E2 -638.061} C_VEL
LIN {X 0,Y 601.386,Z 380.45,A -85,B 0,C 180,E1 -640.992,E2 -640.992} C_VEL
LIN {X 0,Y 601.345,Z 384.416,A -85,B 0,C 180,E1 -643.517,E2 -643.517} C_VEL
LIN {X 0,Y 601.336,Z 388.936,A -85,B 0,C 180,E1 -646.289,E2 -646.289} C_VEL
LIN {X 0,Y 601.309,Z 393.121,A -85,B 0,C 180,E1 -648.788,E2 -648.788} C_VEL
LIN {X 0,Y 601.28,Z 397.314,A -85,B 0,C 180,E1 -651.244,E2 -651.244} C_VEL
LIN {X 0,Y 601.309,Z 401.079,A -85,B 0,C 180,E1 -653.414,E2 -653.414} C_VEL
LIN {X 0,Y 601.343,Z 405.369,A -85,B 0,C 180,E1 -655.853,E2 -655.853} C_VEL
LIN {X 0,Y 601.275,Z 410.562,A -85,B 0,C 180,E1 -658.76,E2 -658.76} C_VEL
LIN {X 0,Y 601.302,Z 414.91,A -85,B 0,C 180,E1 -661.168,E2 -661.168} C_VEL
LIN {X 0,Y 601.604,Z 420.634,A -85,B 0,C 180,E1 -661.294,E2 -661.294} C_VEL
LIN {X 0,Y 601.544,Z 433.296,A -85,B 0,C 180,E1 -661.636,E2 -661.636} C_VEL
LIN {X 0,Y 601.451,Z 445.913,A -85,B 0,C 180,E1 -662.118,E2 -662.118} C_VEL
LIN {X 0,Y 601.425,Z 457.686,A -85,B 0,C 180,E1 -662.716,E2 -662.716} C_VEL
LIN {X 0,Y 601.469,Z 468.412,A -85,B 0,C 180,E1 -663.411,E2 -663.411} C_VEL
LIN {X 0,Y 601.435,Z 478.52,A -85,B 0,C 180,E1 -664.218,E2 -664.218} C_VEL
LIN {X 0,Y 601.419,Z 487.652,A -85,B 0,C 180,E1 -665.115,E2 -665.115} C_VEL
LIN {X 0,Y 601.384,Z 495.059,A -85,B 0,C 180,E1 -666.005,E2 -666.005} C_VEL
LIN {X 0,Y 601.351,Z 501.701,A -85,B 0,C 180,E1 -666.98,E2 -666.98} C_VEL
LIN {X 0,Y 601.349,Z 507.573,A -85,B 0,C 180,E1 -668.06,E2 -668.06} C_VEL
LIN {X 0,Y 601.332,Z 512.074,A -85,B 0,C 180,E1 -669.132,E2 -669.132} C_VEL
LIN {X 0,Y 601.354,Z 514.843,A -85,B 0,C 180,E1 -669.999,E2 -669.999} C_VEL
LIN {X 0,Y 601.317,Z 516.927,A -85,B 0,C 180,E1 -670.882,E2 -670.882} C_VEL
LIN {X 0,Y 601.323,Z 518.263,A -85,B 0,C 180,E1 -671.773,E2 -671.773} C_VEL
LIN {X 0,Y 601.339,Z 518.921,A -85,B 0,C 180,E1 -672.676,E2 -672.676} C_VEL
LIN {X 0,Y 601.341,Z 518.866,A -85,B 0,C 180,E1 -673.593,E2 -673.593} C_VEL
LIN {X 0,Y 601.332,Z 518.019,A -85,B 0,C 180,E1 -674.526,E2 -674.526} C_VEL
LIN {X 0,Y 601.332,Z 516.361,A -85,B 0,C 180,E1 -675.473,E2 -675.473} C_VEL
LIN {X 0,Y 601.343,Z 513.829,A -85,B 0,C 180,E1 -676.435,E2 -676.435} C_VEL
LIN {X 0,Y 601.371,Z 510.324,A -85,B 0,C 180,E1 -677.413,E2 -677.413} C_VEL
LIN {X 0,Y 601.38,Z 505.674,A -85,B 0,C 180,E1 -678.411,E2 -678.411} C_VEL
LIN {X 0,Y 601.355,Z 499.652,A -85,B 0,C 180,E1 -679.432,E2 -679.432} C_VEL
LIN {X 0,Y 601.393,Z 492.024,A -85,B 0,C 180,E1 -680.469,E2 -680.469} C_VEL
LIN {X 0,Y 601.43,Z 483.479,A -85,B 0,C 180,E1 -681.409,E2 -681.409} C_VEL
LIN {X 0,Y 601.456,Z 473.848,A -85,B 0,C 180,E1 -682.266,E2 -682.266} C_VEL
LIN {X 0,Y 601.455,Z 463.703,A -85,B 0,C 180,E1 -683.003,E2 -683.003} C_VEL
LIN {X 0,Y 601.524,Z 452.274,A -85,B 0,C 180,E1 -683.668,E2 -683.668} C_VEL
LIN {X 0,Y 601.53,Z 440.162,A -85,B 0,C 180,E1 -684.21,E2 -684.21} C_VEL
LIN {X 0,Y 601.586,Z 427.31,A -85,B 0,C 180,E1 -684.632,E2 -684.632} C_VEL
LIN {X 0,Y 601.48,Z 416.05,A -85,B 0,C 180,E1 -684.887,E2 -684.887} C_VEL
LIN {X 0,Y 601.332,Z 414.872,A -85,B 0,C 180,E1 -684.943,E2 -684.943} C_VEL
LIN {X 0,Y 601.336,Z 410.292,A -85,B 0,C 180,E1 -687.478,E2 -687.478} C_VEL
LIN {X 0,Y 601.343,Z 404.721,A -85,B 0,C 180,E1 -690.603,E2 -690.603} C_VEL
LIN {X 0,Y 601.351,Z 399.407,A -85,B 0,C 180,E1 -693.634,E2 -693.634} C_VEL
LIN {X 0,Y 601.344,Z 394.332,A -85,B 0,C 180,E1 -696.587,E2 -696.587} C_VEL
LIN {X 0,Y 601.371,Z 389.471,A -85,B 0,C 180,E1 -699.476,E2 -699.476} C_VEL
LIN {X 0,Y 601.366,Z 384.823,A -85,B 0,C 180,E1 -702.311,E2 -702.311} C_VEL
LIN {X 0,Y 601.373,Z 380.508,A -85,B 0,C 180,E1 -705.102,E2 -705.102} C_VEL
LIN {X 0,Y 601.386,Z 377.32,A -85,B 0,C 180,E1 -707.171,E2 -707.171} C_VEL
LIN {X 0,Y 601.41,Z 376.241,A -85,B 0,C 180,E1 -707.857,E2 -707.857} C_VEL
LIN {X 0,Y 601.396,Z 375.575,A -85,B 0,C 180,E1 -708.541,E2 -708.541} C_VEL
LIN {X 0,Y 601.439,Z 375.571,A -85,B 0,C 180,E1 -711.262,E2 -711.262} C_VEL
LIN {X 0,Y 601.406,Z 375.573,A -85,B 0,C 180,E1 -713.963,E2 -713.963} C_VEL
LIN {X 0,Y 601.435,Z 375.572,A -85,B 0,C 180,E1 -716.651,E2 -716.651} C_VEL
LIN {X 0,Y 601.452,Z 375.568,A -85,B 0,C 180,E1 -719.331,E2 -719.331} C_VEL
LIN {X 0,Y 601.423,Z 375.572,A -85,B 0,C 180,E1 -722.009,E2 -722.009} C_VEL
LIN {X 0,Y 601.416,Z 375.573,A -85,B 0,C 180,E1 -724.692,E2 -724.692} C_VEL
LIN {X 0,Y 601.438,Z 375.569,A -85,B 0,C 180,E1 -727.385,E2 -727.385} C_VEL
LIN {X 0,Y 601.431,Z 375.573,A -85,B 0,C 180,E1 -730.095,E2 -730.095} C_VEL
LIN {X 0,Y 601.424,Z 375.571,A -85,B 0,C 180,E1 -732.828,E2 -732.828} C_VEL
LIN {X 0,Y 601.414,Z 375.573,A -85,B 0,C 180,E1 -735.591,E2 -735.591} C_VEL
LIN {X 0,Y 601.398,Z 375.575,A -85,B 0,C 180,E1 -737.688,E2 -737.688} C_VEL
LIN {X 0,Y 601.435,Z 375.572,A -85,B 0,C 180,E1 -740.522,E2 -740.522} C_VEL
LIN {X 0,Y 601.419,Z 375.573,A -85,B 0,C 180,E1 -743.41,E2 -743.41} C_VEL
LIN {X 0,Y 601.401,Z 375.574,A -85,B 0,C 180,E1 -746.364,E2 -746.364} C_VEL
LIN {X 0,Y 601.437,Z 375.572,A -85,B 0,C 180,E1 -748.79,E2 -748.79} C_VEL
LIN {X 0,Y 601.427,Z 375.57,A -85,B 0,C 180,E1 -751.457,E2 -751.457} C_VEL
LIN {X 0,Y 601.43,Z 375.572,A -85,B 0,C 180,E1 -754.118,E2 -754.118} C_VEL
LIN {X 0,Y 601.415,Z 375.572,A -85,B 0,C 180,E1 -756.582,E2 -756.582} C_VEL
LIN {X 0,Y 601.436,Z 375.57,A -85,B 0,C 180,E1 -759.536,E2 -759.536} C_VEL
LIN {X 0,Y 601.416,Z 375.573,A -85,B 0,C 180,E1 -762.592,E2 -762.592} C_VEL
LIN {X 0,Y 601.396,Z 375.577,A -85,B 0,C 180,E1 -765.48,E2 -765.48} C_VEL
LIN {X 0,Y 601.425,Z 375.572,A -85,B 0,C 180,E1 -768.407,E2 -768.407} C_VEL
LIN {X 0,Y 601.432,Z 375.571,A -85,B 0,C 180,E1 -770.876,E2 -770.876} C_VEL
LIN {X 0,Y 601.443,Z 375.571,A -85,B 0,C 180,E1 -773.734,E2 -773.734} C_VEL
LIN {X 0,Y 601.465,Z 375.671,A -85,B 0,C 180,E1 -774.251,E2 -774.251} C_VEL
LIN {X 0,Y 601.528,Z 382.636,A -85,B 0,C 180,E1 -776.693,E2 -776.693} C_VEL
LIN {X 0,Y 601.445,Z 389.798,A -85,B 0,C 180,E1 -779.06,E2 -779.06} C_VEL
LIN {X 0,Y 601.422,Z 396.945,A -85,B 0,C 180,E1 -781.373,E2 -781.373} C_VEL
LIN {X 0,Y 601.465,Z 406.411,A -85,B 0,C 180,E1 -784.384,E2 -784.384} C_VEL
LIN {X 0,Y 601.405,Z 414.695,A -85,B 0,C 180,E1 -786.954,E2 -786.954} C_VEL
LIN {X 0,Y 601.429,Z 424.161,A -85,B 0,C 180,E1 -789.836,E2 -789.836} C_VEL
LIN {X 0,Y 601.388,Z 433.628,A -85,B 0,C 180,E1 -792.663,E2 -792.663} C_VEL
LIN {X 0,Y 601.366,Z 441.911,A -85,B 0,C 180,E1 -795.102,E2 -795.102} C_VEL
LIN {X 0,Y 601.355,Z 451.378,A -85,B 0,C 180,E1 -797.857,E2 -797.857} C_VEL
LIN {X 0,Y 601.379,Z 452.192,A -85,B 0,C 180,E1 -798.092,E2 -798.092} C_VEL
LIN {X 0,Y 601.595,Z 464.196,A -85,B 0,C 180,E1 -798.332,E2 -798.332} C_VEL
LIN {X 0,Y 601.55,Z 476.717,A -85,B 0,C 180,E1 -798.705,E2 -798.705} C_VEL
LIN {X 0,Y 601.482,Z 489.181,A -85,B 0,C 180,E1 -799.225,E2 -799.225} C_VEL
LIN {X 0,Y 601.475,Z 500.174,A -85,B 0,C 180,E1 -799.821,E2 -799.821} C_VEL
LIN {X 0,Y 601.455,Z 511.407,A -85,B 0,C 180,E1 -800.585,E2 -800.585} C_VEL
LIN {X 0,Y 601.423,Z 521.34,A -85,B 0,C 180,E1 -801.432,E2 -801.432} C_VEL
LIN {X 0,Y 601.418,Z 530.963,A -85,B 0,C 180,E1 -802.446,E2 -802.446} C_VEL
LIN {X 0,Y 601.37,Z 538.226,A -85,B 0,C 180,E1 -803.398,E2 -803.398} C_VEL
LIN {X 0,Y 601.372,Z 543.868,A -85,B 0,C 180,E1 -804.299,E2 -804.299} C_VEL
LIN {X 0,Y 601.336,Z 548.951,A -85,B 0,C 180,E1 -805.308,E2 -805.308} C_VEL
LIN {X 0,Y 601.368,Z 552.897,A -85,B 0,C 180,E1 -806.315,E2 -806.315} C_VEL
LIN {X 0,Y 601.325,Z 555.81,A -85,B 0,C 180,E1 -807.321,E2 -807.321} C_VEL
LIN {X 0,Y 601.343,Z 557.202,A -85,B 0,C 180,E1 -807.991,E2 -807.991} C_VEL
LIN {X 0,Y 601.339,Z 558.784,A -85,B 0,C 180,E1 -809.331,E2 -809.331} C_VEL
LIN {X 0,Y 601.335,Z 559,A -85,B 0,C 180,E1 -810,E2 -810} C_VEL
LIN {X 0,Y 601.347,Z 558.184,A -85,B 0,C 180,E1 -811.34,E2 -811.34} C_VEL
LIN {X 0,Y 601.343,Z 557.201,A -85,B 0,C 180,E1 -812.01,E2 -812.01} C_VEL
LIN {X 0,Y 601.325,Z 555.809,A -85,B 0,C 180,E1 -812.68,E2 -812.68} C_VEL
LIN {X 0,Y 601.368,Z 552.895,A -85,B 0,C 180,E1 -813.686,E2 -813.686} C_VEL
LIN {X 0,Y 601.336,Z 548.949,A -85,B 0,C 180,E1 -814.693,E2 -814.693} C_VEL
LIN {X 0,Y 601.372,Z 542.876,A -85,B 0,C 180,E1 -815.869,E2 -815.869} C_VEL
LIN {X 0,Y 601.382,Z 536.234,A -85,B 0,C 180,E1 -816.88,E2 -816.88} C_VEL
LIN {X 0,Y 601.4,Z 527.988,A -85,B 0,C 180,E1 -817.892,E2 -817.892} C_VEL
LIN {X 0,Y 601.436,Z 519.534,A -85,B 0,C 180,E1 -818.738,E2 -818.738} C_VEL
LIN {X 0,Y 601.451,Z 509.089,A -85,B 0,C 180,E1 -819.585,E2 -819.585} C_VEL
LIN {X 0,Y 601.489,Z 498.754,A -85,B 0,C 180,E1 -820.264,E2 -820.264} C_VEL
LIN {X 0,Y 601.491,Z 487.141,A -85,B 0,C 180,E1 -820.873,E2 -820.873} C_VEL
LIN {X 0,Y 601.528,Z 474.314,A -85,B 0,C 180,E1 -821.376,E2 -821.376} C_VEL
LIN {X 0,Y 601.613,Z 461.43,A -85,B 0,C 180,E1 -821.732,E2 -821.732} C_VEL
LIN {X 0,Y 601.38,Z 452.19,A -85,B 0,C 180,E1 -821.908,E2 -821.908} C_VEL
LIN {X 0,Y 601.357,Z 443.093,A -85,B 0,C 180,E1 -824.553,E2 -824.553} C_VEL
LIN {X 0,Y 601.376,Z 434.81,A -85,B 0,C 180,E1 -826.988,E2 -826.988} C_VEL
LIN {X 0,Y 601.413,Z 425.343,A -85,B 0,C 180,E1 -829.809,E2 -829.809} C_VEL
LIN {X 0,Y 601.41,Z 415.876,A -85,B 0,C 180,E1 -832.683,E2 -832.683} C_VEL
LIN {X 0,Y 601.42,Z 407.593,A -85,B 0,C 180,E1 -835.247,E2 -835.247} C_VEL
LIN {X 0,Y 601.443,Z 399.31,A -85,B 0,C 180,E1 -837.866,E2 -837.866} C_VEL
LIN {X 0,Y 601.442,Z 390.999,A -85,B 0,C 180,E1 -840.551,E2 -840.551} C_VEL
LIN {X 0,Y 601.513,Z 384.389,A -85,B 0,C 180,E1 -842.729,E2 -842.729} C_VEL
LIN {X 0,Y 601.549,Z 377.405,A -85,B 0,C 180,E1 -845.132,E2 -845.132} C_VEL
LIN {X 0,Y 601.441,Z 375.57,A -85,B 0,C 180,E1 -845.841,E2 -845.841} C_VEL
LIN {X 0,Y 601.413,Z 375.573,A -85,B 0,C 180,E1 -848.468,E2 -848.468} C_VEL
LIN {X 0,Y 601.414,Z 375.573,A -85,B 0,C 180,E1 -850.874,E2 -850.874} C_VEL
LIN {X 0,Y 601.429,Z 375.573,A -85,B 0,C 180,E1 -853.586,E2 -853.586} C_VEL
LIN {X 0,Y 601.43,Z 375.569,A -85,B 0,C 180,E1 -856.427,E2 -856.427} C_VEL
LIN {X 0,Y 601.405,Z 375.573,A -85,B 0,C 180,E1 -859.125,E2 -859.125} C_VEL
LIN {X 0,Y 601.426,Z 375.572,A -85,B 0,C 180,E1 -861.732,E2 -861.732} C_VEL
LIN {X 0,Y 601.397,Z 375.577,A -85,B 0,C 180,E1 -864.246,E2 -864.246} C_VEL
LIN {X 0,Y 601.419,Z 375.574,A -85,B 0,C 180,E1 -866.686,E2 -866.686} C_VEL
LIN {X 0,Y 601.414,Z 375.575,A -85,B 0,C 180,E1 -869.058,E2 -869.058} C_VEL
LIN {X 0,Y 601.433,Z 375.572,A -85,B 0,C 180,E1 -871.373,E2 -871.373} C_VEL
LIN {X 0,Y 601.401,Z 375.575,A -85,B 0,C 180,E1 -873.636,E2 -873.636} C_VEL
LIN {X 0,Y 601.42,Z 375.571,A -85,B 0,C 180,E1 -876.59,E2 -876.59} C_VEL
LIN {X 0,Y 601.435,Z 375.57,A -85,B 0,C 180,E1 -879.478,E2 -879.478} C_VEL
LIN {X 0,Y 601.395,Z 375.576,A -85,B 0,C 180,E1 -882.312,E2 -882.312} C_VEL
LIN {X 0,Y 601.41,Z 375.574,A -85,B 0,C 180,E1 -884.409,E2 -884.409} C_VEL
LIN {X 0,Y 601.415,Z 375.572,A -85,B 0,C 180,E1 -887.172,E2 -887.172} C_VEL
LIN {X 0,Y 601.424,Z 375.57,A -85,B 0,C 180,E1 -889.905,E2 -889.905} C_VEL
LIN {X 0,Y 601.44,Z 375.569,A -85,B 0,C 180,E1 -892.615,E2 -892.615} C_VEL
LIN {X 0,Y 601.422,Z 375.574,A -85,B 0,C 180,E1 -895.308,E2 -895.308} C_VEL
LIN {X 0,Y 601.414,Z 375.572,A -85,B 0,C 180,E1 -897.991,E2 -897.991} C_VEL
LIN {X 0,Y 601.446,Z 375.567,A -85,B 0,C 180,E1 -900.669,E2 -900.669} C_VEL
LIN {X 0,Y 601.433,Z 375.57,A -85,B 0,C 180,E1 -903.35,E2 -903.35} C_VEL
LIN {X 0,Y 601.415,Z 375.575,A -85,B 0,C 180,E1 -906.037,E2 -906.037} C_VEL
LIN {X 0,Y 601.44,Z 375.569,A -85,B 0,C 180,E1 -908.738,E2 -908.738} C_VEL
LIN {X 0,Y 601.422,Z 375.57,A -85,B 0,C 180,E1 -911.458,E2 -911.458} C_VEL
LIN {X 0,Y 601.408,Z 375.572,A -85,B 0,C 180,E1 -912.371,E2 -912.371} C_VEL
LIN {X 0,Y 600.743,Z 375.657,A -85,B 0,C 180,E1 -912.93,E2 -912.93} C_VEL
LIN {X 0,Y 597.896,Z 376.009,A -85,B 0,C 180,E1 -913.838,E2 -913.838} C_VEL
LIN {X 0,Y 595.487,Z 376.311,A -85,B 0,C 180,E1 -914.569,E2 -914.569} C_VEL
LIN {X 0,Y 594.447,Z 376.439,A -85,B 0,C 180,E1 -915.132,E2 -915.132} C_VEL
LIN {X 0,Y 594.36,Z 376.449,A -85,B 0,C 180,E1 -915.323,E2 -915.323} C_VEL
LIN {X 0,Y 594.378,Z 376.451,A -85,B 0,C 180,E1 -917.904,E2 -917.904} C_VEL
LIN {X 0,Y 594.385,Z 376.447,A -85,B 0,C 180,E1 -920.918,E2 -920.918} C_VEL
LIN {X 0,Y 594.39,Z 376.448,A -85,B 0,C 180,E1 -923.704,E2 -923.704} C_VEL
LIN {X 0,Y 594.385,Z 376.447,A -85,B 0,C 180,E1 -926.7,E2 -926.7} C_VEL
LIN {X 0,Y 594.377,Z 376.448,A -85,B 0,C 180,E1 -928.999,E2 -928.999} C_VEL
LIN {X 0,Y 594.377,Z 376.447,A -85,B 0,C 180,E1 -931.643,E2 -931.643} C_VEL
LIN {X 0,Y 594.38,Z 376.45,A -85,B 0,C 180,E1 -934.58,E2 -934.58} C_VEL
LIN {X 0,Y 594.388,Z 376.449,A -85,B 0,C 180,E1 -937.087,E2 -937.087} C_VEL
LIN {X 0,Y 594.356,Z 376.451,A -85,B 0,C 180,E1 -939.772,E2 -939.772} C_VEL
LIN {X 0,Y 594.371,Z 376.449,A -85,B 0,C 180,E1 -942.375,E2 -942.375} C_VEL
LIN {X 0,Y 594.345,Z 376.454,A -85,B 0,C 180,E1 -945.193,E2 -945.193} C_VEL
LIN {X 0,Y 594.388,Z 376.447,A -85,B 0,C 180,E1 -948.151,E2 -948.151} C_VEL
LIN {X 0,Y 594.373,Z 376.452,A -85,B 0,C 180,E1 -951.297,E2 -951.297} C_VEL
LIN {X 0,Y 594.395,Z 376.449,A -85,B 0,C 180,E1 -953.759,E2 -953.759} C_VEL
LIN {X 0,Y 594.379,Z 376.45,A -85,B 0,C 180,E1 -956.239,E2 -956.239} C_VEL
LIN {X 0,Y 594.369,Z 376.451,A -85,B 0,C 180,E1 -958.65,E2 -958.65} C_VEL
LIN {X 0,Y 594.382,Z 376.449,A -85,B 0,C 180,E1 -961.043,E2 -961.043} C_VEL
LIN {X 0,Y 594.393,Z 376.446,A -85,B 0,C 180,E1 -963.976,E2 -963.976} C_VEL
LIN {X 0,Y 594.392,Z 376.446,A -85,B 0,C 180,E1 -966.296,E2 -966.296} C_VEL
LIN {X 0,Y 594.404,Z 376.448,A -85,B 0,C 180,E1 -969.224,E2 -969.224} C_VEL
LIN {X 0,Y 594.359,Z 376.45,A -85,B 0,C 180,E1 -972.095,E2 -972.095} C_VEL
LIN {X 0,Y 594.363,Z 376.451,A -85,B 0,C 180,E1 -974.219,E2 -974.219} C_VEL
LIN {X 0,Y 594.381,Z 376.45,A -85,B 0,C 180,E1 -976.321,E2 -976.321} C_VEL
LIN {X 0,Y 594.368,Z 376.449,A -85,B 0,C 180,E1 -979.094,E2 -979.094} C_VEL
LIN {X 0,Y 594.417,Z 376.443,A -85,B 0,C 180,E1 -981.843,E2 -981.843} C_VEL
LIN {X 0,Y 594.401,Z 376.447,A -85,B 0,C 180,E1 -984.572,E2 -984.572} C_VEL
LIN {X 0,Y 594.407,Z 376.446,A -85,B 0,C 180,E1 -987.289,E2 -987.289} C_VEL
LIN {X 0,Y 594.419,Z 376.443,A -85,B 0,C 180,E1 -990,E2 -990} C_VEL
LIN {X 0,Y 594.4,Z 376.445,A -85,B 0,C 180,E1 -992.711,E2 -992.711} C_VEL
LIN {X 0,Y 594.391,Z 376.449,A -85,B 0,C 180,E1 -995.427,E2 -995.427} C_VEL
LIN {X 0,Y 594.352,Z 376.451,A -85,B 0,C 180,E1 -997.473,E2 -997.473} C_VEL
LIN {X 0,Y 594.342,Z 376.819,A -85,B 0,C 180,E1 -998.157,E2 -998.157} C_VEL
LIN {X 0,Y 594.331,Z 381.242,A -85,B 0,C 180,E1 -1001.043,E2 -1001.043} C_VEL
LIN {X 0,Y 594.301,Z 385.395,A -85,B 0,C 180,E1 -1003.68,E2 -1003.68} C_VEL
LIN {X 0,Y 594.256,Z 389.826,A -85,B 0,C 180,E1 -1006.489,E2 -1006.489} C_VEL
LIN {X 0,Y 594.226,Z 394.557,A -85,B 0,C 180,E1 -1009.339,E2 -1009.339} C_VEL
LIN {X 0,Y 594.206,Z 398.231,A -85,B 0,C 180,E1 -1011.509,E2 -1011.509} C_VEL
LIN {X 0,Y 594.232,Z 403.297,A -85,B 0,C 180,E1 -1014.452,E2 -1014.452} C_VEL
LIN {X 0,Y 594.211,Z 407.241,A -85,B 0,C 180,E1 -1016.707,E2 -1016.707} C_VEL
LIN {X 0,Y 594.197,Z 412.696,A -85,B 0,C 180,E1 -1019.786,E2 -1019.786} C_VEL
LIN {X 0,Y 594.213,Z 415.075,A -85,B 0,C 180,E1 -1021.037,E2 -1021.037} C_VEL
LIN {X 0,Y 594.67,Z 420.274,A -85,B 0,C 180,E1 -1021.146,E2 -1021.146} C_VEL
LIN {X 0,Y 594.573,Z 433.624,A -85,B 0,C 180,E1 -1021.511,E2 -1021.511} C_VEL
LIN {X 0,Y 594.486,Z 446.29,A -85,B 0,C 180,E1 -1022.005,E2 -1022.005} C_VEL
LIN {X 0,Y 594.425,Z 458.543,A -85,B 0,C 180,E1 -1022.644,E2 -1022.644} C_VEL
LIN {X 0,Y 594.447,Z 469.147,A -85,B 0,C 180,E1 -1023.35,E2 -1023.35} C_VEL
LIN {X 0,Y 594.407,Z 479.39,A -85,B 0,C 180,E1 -1024.19,E2 -1024.19} C_VEL
LIN {X 0,Y 594.333,Z 488.845,A -85,B 0,C 180,E1 -1025.157,E2 -1025.157} C_VEL
LIN {X 0,Y 594.32,Z 497.415,A -85,B 0,C 180,E1 -1026.246,E2 -1026.246} C_VEL
LIN {X 0,Y 594.294,Z 504.215,A -85,B 0,C 180,E1 -1027.341,E2 -1027.341} C_VEL
LIN {X 0,Y 594.253,Z 509.045,A -85,B 0,C 180,E1 -1028.319,E2 -1028.319} C_VEL
LIN {X 0,Y 594.239,Z 512.68,A -85,B 0,C 180,E1 -1029.252,E2 -1029.252} C_VEL
LIN {X 0,Y 594.255,Z 515.313,A -85,B 0,C 180,E1 -1030.142,E2 -1030.142} C_VEL
LIN {X 0,Y 594.217,Z 516.818,A -85,B 0,C 180,E1 -1030.804,E2 -1030.804} C_VEL
LIN {X 0,Y 594.246,Z 518.35,A -85,B 0,C 180,E1 -1031.834,E2 -1031.834} C_VEL
LIN {X 0,Y 594.245,Z 518.959,A -85,B 0,C 180,E1 -1032.84,E2 -1032.84} C_VEL
LIN {X 0,Y 594.228,Z 518.357,A -85,B 0,C 180,E1 -1034.25,E2 -1034.25} C_VEL
LIN {X 0,Y 594.258,Z 516.992,A -85,B 0,C 180,E1 -1035.201,E2 -1035.201} C_VEL
LIN {X 0,Y 594.248,Z 514.727,A -85,B 0,C 180,E1 -1036.172,E2 -1036.172} C_VEL
LIN {X 0,Y 594.269,Z 511.52,A -85,B 0,C 180,E1 -1037.157,E2 -1037.157} C_VEL
LIN {X 0,Y 594.284,Z 507.233,A -85,B 0,C 180,E1 -1038.161,E2 -1038.161} C_VEL
LIN {X 0,Y 594.262,Z 501.659,A -85,B 0,C 180,E1 -1039.19,E2 -1039.19} C_VEL
LIN {X 0,Y 594.323,Z 493.952,A -85,B 0,C 180,E1 -1040.315,E2 -1040.315} C_VEL
LIN {X 0,Y 594.358,Z 485.506,A -85,B 0,C 180,E1 -1041.298,E2 -1041.298} C_VEL
LIN {X 0,Y 594.405,Z 476.492,A -85,B 0,C 180,E1 -1042.156,E2 -1042.156} C_VEL
LIN {X 0,Y 594.445,Z 465.534,A -85,B 0,C 180,E1 -1042.998,E2 -1042.998} C_VEL
LIN {X 0,Y 594.521,Z 453.992,A -85,B 0,C 180,E1 -1043.701,E2 -1043.701} C_VEL
LIN {X 0,Y 594.563,Z 442.694,A -85,B 0,C 180,E1 -1044.241,E2 -1044.241} C_VEL
LIN {X 0,Y 594.603,Z 429.928,A -85,B 0,C 180,E1 -1044.696,E2 -1044.696} C_VEL
LIN {X 0,Y 594.553,Z 416.865,A -85,B 0,C 180,E1 -1045.012,E2 -1045.012} C_VEL
LIN {X 0,Y 594.283,Z 414.904,A -85,B 0,C 180,E1 -1045.068,E2 -1045.068} C_VEL
LIN {X 0,Y 594.235,Z 409.955,A -85,B 0,C 180,E1 -1047.845,E2 -1047.845} C_VEL
LIN {X 0,Y 594.239,Z 405.776,A -85,B 0,C 180,E1 -1050.216,E2 -1050.216} C_VEL
LIN {X 0,Y 594.257,Z 401.743,A -85,B 0,C 180,E1 -1052.533,E2 -1052.533} C_VEL
LIN {X 0,Y 594.263,Z 397.851,A -85,B 0,C 180,E1 -1054.802,E2 -1054.802} C_VEL
LIN {X 0,Y 594.273,Z 392.863,A -85,B 0,C 180,E1 -1057.763,E2 -1057.763} C_VEL
LIN {X 0,Y 594.272,Z 389.265,A -85,B 0,C 180,E1 -1059.943,E2 -1059.943} C_VEL
LIN {X 0,Y 594.297,Z 385.907,A -85,B 0,C 180,E1 -1062.093,E2 -1062.093} C_VEL
LIN {X 0,Y 594.302,Z 382.625,A -85,B 0,C 180,E1 -1064.217,E2 -1064.217} C_VEL
LIN {X 0,Y 594.36,Z 379.389,A -85,B 0,C 180,E1 -1066.321,E2 -1066.321} C_VEL
LIN {X 0,Y 594.343,Z 377.232,A -85,B 0,C 180,E1 -1067.711,E2 -1067.711} C_VEL
LIN {X 0,Y 594.347,Z 376.454,A -85,B 0,C 180,E1 -1068.403,E2 -1068.403} C_VEL
LIN {X 0,Y 594.399,Z 376.447,A -85,B 0,C 180,E1 -1071.158,E2 -1071.158} C_VEL
LIN {X 0,Y 594.363,Z 376.451,A -85,B 0,C 180,E1 -1073.891,E2 -1073.891} C_VEL
LIN {X 0,Y 594.386,Z 376.45,A -85,B 0,C 180,E1 -1076.611,E2 -1076.611} C_VEL
LIN {X 0,Y 594.423,Z 376.443,A -85,B 0,C 180,E1 -1079.323,E2 -1079.323} C_VEL
LIN {X 0,Y 594.393,Z 376.447,A -85,B 0,C 180,E1 -1082.033,E2 -1082.033} C_VEL
LIN {X 0,Y 594.386,Z 376.449,A -85,B 0,C 180,E1 -1084.748,E2 -1084.748} C_VEL
LIN {X 0,Y 594.391,Z 376.447,A -85,B 0,C 180,E1 -1087.473,E2 -1087.473} C_VEL
LIN {X 0,Y 594.392,Z 376.448,A -85,B 0,C 180,E1 -1090.216,E2 -1090.216} C_VEL
LIN {X 0,Y 594.371,Z 376.45,A -85,B 0,C 180,E1 -1092.983,E2 -1092.983} C_VEL
LIN {X 0,Y 594.367,Z 376.45,A -85,B 0,C 180,E1 -1095.781,E2 -1095.781} C_VEL
LIN {X 0,Y 594.386,Z 376.449,A -85,B 0,C 180,E1 -1098.617,E2 -1098.617} C_VEL
LIN {X 0,Y 594.368,Z 376.452,A -85,B 0,C 180,E1 -1101.503,E2 -1101.503} C_VEL
LIN {X 0,Y 594.384,Z 376.449,A -85,B 0,C 180,E1 -1104.446,E2 -1104.446} C_VEL
LIN {X 0,Y 594.381,Z 376.451,A -85,B 0,C 180,E1 -1106.7,E2 -1106.7} C_VEL
LIN {X 0,Y 594.38,Z 376.45,A -85,B 0,C 180,E1 -1108.999,E2 -1108.999} C_VEL
LIN {X 0,Y 594.382,Z 376.449,A -85,B 0,C 180,E1 -1111.644,E2 -1111.644} C_VEL
LIN {X 0,Y 594.382,Z 376.448,A -85,B 0,C 180,E1 -1114.58,E2 -1114.58} C_VEL
LIN {X 0,Y 594.386,Z 376.45,A -85,B 0,C 180,E1 -1117.087,E2 -1117.087} C_VEL
LIN {X 0,Y 594.373,Z 376.449,A -85,B 0,C 180,E1 -1119.775,E2 -1119.775} C_VEL
LIN {X 0,Y 594.371,Z 376.452,A -85,B 0,C 180,E1 -1122.375,E2 -1122.375} C_VEL
LIN {X 0,Y 594.362,Z 376.451,A -85,B 0,C 180,E1 -1125.192,E2 -1125.192} C_VEL
LIN {X 0,Y 594.382,Z 376.448,A -85,B 0,C 180,E1 -1128.152,E2 -1128.152} C_VEL
LIN {X 0,Y 594.385,Z 376.448,A -85,B 0,C 180,E1 -1131.196,E2 -1131.196} C_VEL
LIN {X 0,Y 594.418,Z 376.552,A -85,B 0,C 180,E1 -1134.075,E2 -1134.075} C_VEL
LIN {X 0,Y 594.541,Z 382.606,A -85,B 0,C 180,E1 -1136.25,E2 -1136.25} C_VEL
LIN {X 0,Y 594.44,Z 390.922,A -85,B 0,C 180,E1 -1139.05,E2 -1139.05} C_VEL
LIN {X 0,Y 594.431,Z 398.167,A -85,B 0,C 180,E1 -1141.404,E2 -1141.404} C_VEL
LIN {X 0,Y 594.429,Z 407.595,A -85,B 0,C 180,E1 -1144.435,E2 -1144.435} C_VEL
LIN {X 0,Y 594.365,Z 415.878,A -85,B 0,C 180,E1 -1147.033,E2 -1147.033} C_VEL
LIN {X 0,Y 594.384,Z 424.161,A -85,B 0,C 180,E1 -1149.586,E2 -1149.586} C_VEL
LIN {X 0,Y 594.327,Z 433.628,A -85,B 0,C 180,E1 -1152.45,E2 -1152.45} C_VEL
LIN {X 0,Y 594.301,Z 443.095,A -85,B 0,C 180,E1 -1155.271,E2 -1155.271} C_VEL
LIN {X 0,Y 594.288,Z 452.192,A -85,B 0,C 180,E1 -1157.948,E2 -1157.948} C_VEL
LIN {X 0,Y 594.675,Z 457.248,A -85,B 0,C 180,E1 -1158.043,E2 -1158.043} C_VEL
LIN {X 0,Y 594.613,Z 470.509,A -85,B 0,C 180,E1 -1158.366,E2 -1158.366} C_VEL
LIN {X 0,Y 594.536,Z 482.982,A -85,B 0,C 180,E1 -1158.816,E2 -1158.816} C_VEL
LIN {X 0,Y 594.486,Z 495.782,A -85,B 0,C 180,E1 -1159.442,E2 -1159.442} C_VEL
LIN {X 0,Y 594.46,Z 506.752,A -85,B 0,C 180,E1 -1160.13,E2 -1160.13} C_VEL
LIN {X 0,Y 594.404,Z 517.603,A -85,B 0,C 180,E1 -1160.987,E2 -1160.987} C_VEL
LIN {X 0,Y 594.365,Z 526.416,A -85,B 0,C 180,E1 -1161.843,E2 -1161.843} C_VEL
LIN {X 0,Y 594.304,Z 535.001,A -85,B 0,C 180,E1 -1162.868,E2 -1162.868} C_VEL
LIN {X 0,Y 594.289,Z 541.868,A -85,B 0,C 180,E1 -1163.891,E2 -1163.891} C_VEL
LIN {X 0,Y 594.254,Z 547.367,A -85,B 0,C 180,E1 -1164.912,E2 -1164.912} C_VEL
LIN {X 0,Y 594.263,Z 551.678,A -85,B 0,C 180,E1 -1165.931,E2 -1165.931} C_VEL
LIN {X 0,Y 594.267,Z 553.957,A -85,B 0,C 180,E1 -1166.61,E2 -1166.61} C_VEL
LIN {X 0,Y 594.226,Z 555.81,A -85,B 0,C 180,E1 -1167.289,E2 -1167.289} C_VEL
LIN {X 0,Y 594.242,Z 557.202,A -85,B 0,C 180,E1 -1167.967,E2 -1167.967} C_VEL
LIN {X 0,Y 594.239,Z 558.784,A -85,B 0,C 180,E1 -1169.323,E2 -1169.323} C_VEL
LIN {X 0,Y 594.236,Z 559,A -85,B 0,C 180,E1 -1170,E2 -1170} C_VEL
LIN {X 0,Y 594.247,Z 558.184,A -85,B 0,C 180,E1 -1171.356,E2 -1171.356} C_VEL
LIN {X 0,Y 594.242,Z 557.201,A -85,B 0,C 180,E1 -1172.034,E2 -1172.034} C_VEL
LIN {X 0,Y 594.226,Z 555.809,A -85,B 0,C 180,E1 -1172.712,E2 -1172.712} C_VEL
LIN {X 0,Y 594.289,Z 552.895,A -85,B 0,C 180,E1 -1173.73,E2 -1173.73} C_VEL
LIN {X 0,Y 594.241,Z 548.949,A -85,B 0,C 180,E1 -1174.749,E2 -1174.749} C_VEL
LIN {X 0,Y 594.304,Z 542.876,A -85,B 0,C 180,E1 -1175.939,E2 -1175.939} C_VEL
LIN {X 0,Y 594.308,Z 536.234,A -85,B 0,C 180,E1 -1176.962,E2 -1176.962} C_VEL
LIN {X 0,Y 594.359,Z 527.988,A -85,B 0,C 180,E1 -1177.987,E2 -1177.987} C_VEL
LIN {X 0,Y 594.382,Z 519.535,A -85,B 0,C 180,E1 -1178.842,E2 -1178.842} C_VEL
LIN {X 0,Y 594.434,Z 509.091,A -85,B 0,C 180,E1 -1179.7,E2 -1179.7} C_VEL
LIN {X 0,Y 594.464,Z 498.755,A -85,B 0,C 180,E1 -1180.387,E2 -1180.387} C_VEL
LIN {X 0,Y 594.506,Z 486.717,A -85,B 0,C 180,E1 -1181.021,E2 -1181.021} C_VEL
LIN {X 0,Y 594.565,Z 474.48,A -85,B 0,C 180,E1 -1181.506,E2 -1181.506} C_VEL
LIN {X 0,Y 594.67,Z 461.43,A -85,B 0,C 180,E1 -1181.871,E2 -1181.871} C_VEL
LIN {X 0,Y 594.492,Z 453.601,A -85,B 0,C 180,E1 -1182.026,E2 -1182.026} C_VEL
LIN {X 0,Y 594.293,Z 452.116,A -85,B 0,C 180,E1 -1182.074,E2 -1182.074} C_VEL
LIN {X 0,Y 594.301,Z 443.093,A -85,B 0,C 180,E1 -1184.729,E2 -1184.729} C_VEL
LIN {X 0,Y 594.327,Z 433.626,A -85,B 0,C 180,E1 -1187.55,E2 -1187.55} C_VEL
LIN {X 0,Y 594.385,Z 424.16,A -85,B 0,C 180,E1 -1190.415,E2 -1190.415} C_VEL
LIN {X 0,Y 594.377,Z 414.693,A -85,B 0,C 180,E1 -1193.335,E2 -1193.335} C_VEL
LIN {X 0,Y 594.424,Z 405.206,A -85,B 0,C 180,E1 -1196.326,E2 -1196.326} C_VEL
LIN {X 0,Y 594.47,Z 395.733,A -85,B 0,C 180,E1 -1199.382,E2 -1199.382} C_VEL
LIN {X 0,Y 594.501,Z 386.199,A -85,B 0,C 180,E1 -1202.535,E2 -1202.535} C_VEL
LIN {X 0,Y 594.542,Z 379.221,A -85,B 0,C 180,E1 -1204.959,E2 -1204.959} C_VEL
LIN {X 0,Y 594.384,Z 376.45,A -85,B 0,C 180,E1 -1206.032,E2 -1206.032} C_VEL
LIN {X 0,Y 594.38,Z 376.451,A -85,B 0,C 180,E1 -1208.805,E2 -1208.805} C_VEL
LIN {X 0,Y 594.385,Z 376.447,A -85,B 0,C 180,E1 -1211.848,E2 -1211.848} C_VEL
LIN {X 0,Y 594.346,Z 376.454,A -85,B 0,C 180,E1 -1214.807,E2 -1214.807} C_VEL
LIN {X 0,Y 594.37,Z 376.449,A -85,B 0,C 180,E1 -1217.624,E2 -1217.624} C_VEL
LIN {X 0,Y 594.37,Z 376.449,A -85,B 0,C 180,E1 -1220.319,E2 -1220.319} C_VEL
LIN {X 0,Y 594.385,Z 376.449,A -85,B 0,C 180,E1 -1222.913,E2 -1222.913} C_VEL
LIN {X 0,Y 594.372,Z 376.448,A -85,B 0,C 180,E1 -1225.863,E2 -1225.863} C_VEL
LIN {X 0,Y 594.369,Z 376.449,A -85,B 0,C 180,E1 -1228.65,E2 -1228.65} C_VEL
LIN {X 0,Y 594.384,Z 376.447,A -85,B 0,C 180,E1 -1231.042,E2 -1231.042} C_VEL
LIN {X 0,Y 594.386,Z 376.447,A -85,B 0,C 180,E1 -1233.3,E2 -1233.3} C_VEL
LIN {X 0,Y 594.389,Z 376.449,A -85,B 0,C 180,E1 -1236.296,E2 -1236.296} C_VEL
LIN {X 0,Y 594.409,Z 376.444,A -85,B 0,C 180,E1 -1239.225,E2 -1239.225} C_VEL
LIN {X 0,Y 594.354,Z 376.454,A -85,B 0,C 180,E1 -1242.095,E2 -1242.095} C_VEL
LIN {X 0,Y 594.362,Z 376.45,A -85,B 0,C 180,E1 -1244.219,E2 -1244.219} C_VEL
LIN {X 0,Y 594.378,Z 376.447,A -85,B 0,C 180,E1 -1246.321,E2 -1246.321} C_VEL
LIN {X 0,Y 594.378,Z 376.449,A -85,B 0,C 180,E1 -1249.095,E2 -1249.095} C_VEL
LIN {X 0,Y 594.411,Z 376.446,A -85,B 0,C 180,E1 -1251.843,E2 -1251.843} C_VEL
LIN {X 0,Y 594.392,Z 376.446,A -85,B 0,C 180,E1 -1254.572,E2 -1254.572} C_VEL
LIN {X 0,Y 594.413,Z 376.444,A -85,B 0,C 180,E1 -1257.289,E2 -1257.289} C_VEL
LIN {X 0,Y 594.414,Z 376.446,A -85,B 0,C 180,E1 -1260,E2 -1260} C_VEL
LIN {X 0,Y 594.414,Z 376.444,A -85,B 0,C 180,E1 -1262.711,E2 -1262.711} C_VEL
LIN {X 0,Y 594.389,Z 376.446,A -85,B 0,C 180,E1 -1265.428,E2 -1265.428} C_VEL
LIN {X 0,Y 594.411,Z 376.445,A -85,B 0,C 180,E1 -1268.157,E2 -1268.157} C_VEL
LIN {X 0,Y 594.391,Z 376.447,A -85,B 0,C 180,E1 -1271.075,E2 -1271.075} C_VEL
LIN {X 0,Y 594.38,Z 376.447,A -85,B 0,C 180,E1 -1273.679,E2 -1273.679} C_VEL
LIN {X 0,Y 594.36,Z 376.449,A -85,B 0,C 180,E1 -1275.323,E2 -1275.323} C_VEL
LIN {X 0,Y 593.686,Z 376.535,A -85,B 0,C 180,E1 -1275.889,E2 -1275.889} C_VEL
LIN {X 0,Y 590.832,Z 376.892,A -85,B 0,C 180,E1 -1276.807,E2 -1276.807} C_VEL
LIN {X 0,Y 588.43,Z 377.192,A -85,B 0,C 180,E1 -1277.546,E2 -1277.546} C_VEL
LIN {X 0,Y 587.404,Z 377.318,A -85,B 0,C 180,E1 -1278.116,E2 -1278.116} C_VEL
LIN {X 0,Y 587.323,Z 377.327,A -85,B 0,C 180,E1 -1278.309,E2 -1278.309} C_VEL
LIN {X 0,Y 587.331,Z 377.326,A -85,B 0,C 180,E1 -1281.038,E2 -1281.038} C_VEL
LIN {X 0,Y 587.337,Z 377.327,A -85,B 0,C 180,E1 -1284.006,E2 -1284.006} C_VEL
LIN {X 0,Y 587.336,Z 377.328,A -85,B 0,C 180,E1 -1286.279,E2 -1286.279} C_VEL
LIN {X 0,Y 587.347,Z 377.324,A -85,B 0,C 180,E1 -1289.133,E2 -1289.133} C_VEL
LIN {X 0,Y 587.345,Z 377.324,A -85,B 0,C 180,E1 -1291.836,E2 -1291.836} C_VEL
LIN {X 0,Y 587.348,Z 377.324,A -85,B 0,C 180,E1 -1294.348,E2 -1294.348} C_VEL
LIN {X 0,Y 587.355,Z 377.324,A -85,B 0,C 180,E1 -1296.747,E2 -1296.747} C_VEL
LIN {X 0,Y 587.331,Z 377.329,A -85,B 0,C 180,E1 -1299.361,E2 -1299.361} C_VEL
LIN {X 0,Y 587.336,Z 377.326,A -85,B 0,C 180,E1 -1302.108,E2 -1302.108} C_VEL
LIN {X 0,Y 587.301,Z 377.33,A -85,B 0,C 180,E1 -1305.087,E2 -1305.087} C_VEL
LIN {X 0,Y 587.355,Z 377.325,A -85,B 0,C 180,E1 -1307.928,E2 -1307.928} C_VEL
LIN {X 0,Y 587.319,Z 377.328,A -85,B 0,C 180,E1 -1311.06,E2 -1311.06} C_VEL
LIN {X 0,Y 587.354,Z 377.323,A -85,B 0,C 180,E1 -1313.292,E2 -1313.292} C_VEL
LIN {X 0,Y 587.359,Z 377.322,A -85,B 0,C 180,E1 -1315.78,E2 -1315.78} C_VEL
LIN {X 0,Y 587.341,Z 377.325,A -85,B 0,C 180,E1 -1318.231,E2 -1318.231} C_VEL
LIN {X 0,Y 587.35,Z 377.327,A -85,B 0,C 180,E1 -1320.867,E2 -1320.867} C_VEL
LIN {X 0,Y 587.364,Z 377.321,A -85,B 0,C 180,E1 -1323.818,E2 -1323.818} C_VEL
LIN {X 0,Y 587.339,Z 377.325,A -85,B 0,C 180,E1 -1325.994,E2 -1325.994} C_VEL
LIN {X 0,Y 587.334,Z 377.326,A -85,B 0,C 180,E1 -1328.962,E2 -1328.962} C_VEL
LIN {X 0,Y 587.348,Z 377.323,A -85,B 0,C 180,E1 -1331.151,E2 -1331.151} C_VEL
LIN {X 0,Y 587.318,Z 377.331,A -85,B 0,C 180,E1 -1334.024,E2 -1334.024} C_VEL
LIN {X 0,Y 587.36,Z 377.323,A -85,B 0,C 180,E1 -1336.154,E2 -1336.154} C_VEL
LIN {X 0,Y 587.34,Z 377.326,A -85,B 0,C 180,E1 -1338.962,E2 -1338.962} C_VEL
LIN {X 0,Y 587.368,Z 377.321,A -85,B 0,C 180,E1 -1341.745,E2 -1341.745} C_VEL
LIN {X 0,Y 587.366,Z 377.323,A -85,B 0,C 180,E1 -1344.507,E2 -1344.507} C_VEL
LIN {X 0,Y 587.373,Z 377.323,A -85,B 0,C 180,E1 -1347.257,E2 -1347.257} C_VEL
LIN {X 0,Y 587.388,Z 377.319,A -85,B 0,C 180,E1 -1350,E2 -1350} C_VEL
LIN {X 0,Y 587.367,Z 377.322,A -85,B 0,C 180,E1 -1352.743,E2 -1352.743} C_VEL
LIN {X 0,Y 587.358,Z 377.326,A -85,B 0,C 180,E1 -1355.493,E2 -1355.493} C_VEL
LIN {X 0,Y 587.31,Z 377.329,A -85,B 0,C 180,E1 -1357.564,E2 -1357.564} C_VEL
LIN {X 0,Y 587.272,Z 377.714,A -85,B 0,C 180,E1 -1358.256,E2 -1358.256} C_VEL
LIN {X 0,Y 587.282,Z 382.037,A -85,B 0,C 180,E1 -1361.099,E2 -1361.099} C_VEL
LIN {X 0,Y 587.263,Z 386.923,A -85,B 0,C 180,E1 -1364.22,E2 -1364.22} C_VEL
LIN {X 0,Y 587.177,Z 390.822,A -85,B 0,C 180,E1 -1366.758,E2 -1366.758} C_VEL
LIN {X 0,Y 587.157,Z 395.462,A -85,B 0,C 180,E1 -1369.581,E2 -1369.581} C_VEL
LIN {X 0,Y 587.131,Z 400.402,A -85,B 0,C 180,E1 -1372.522,E2 -1372.522} C_VEL
LIN {X 0,Y 587.153,Z 404.236,A -85,B 0,C 180,E1 -1374.767,E2 -1374.767} C_VEL
LIN {X 0,Y 587.131,Z 409.237,A -85,B 0,C 180,E1 -1377.651,E2 -1377.651} C_VEL
LIN {X 0,Y 587.111,Z 414.547,A -85,B 0,C 180,E1 -1380.671,E2 -1380.671} C_VEL
LIN {X 0,Y 587.103,Z 414.922,A -85,B 0,C 180,E1 -1380.883,E2 -1380.883} C_VEL
LIN {X 0,Y 587.714,Z 420.382,A -85,B 0,C 180,E1 -1381.006,E2 -1381.006} C_VEL
LIN {X 0,Y 587.636,Z 432.897,A -85,B 0,C 180,E1 -1381.348,E2 -1381.348} C_VEL
LIN {X 0,Y 587.509,Z 446.049,A -85,B 0,C 180,E1 -1381.861,E2 -1381.861} C_VEL
LIN {X 0,Y 587.408,Z 457.856,A -85,B 0,C 180,E1 -1382.477,E2 -1382.477} C_VEL
LIN {X 0,Y 587.418,Z 469.011,A -85,B 0,C 180,E1 -1383.222,E2 -1383.222} C_VEL
LIN {X 0,Y 587.364,Z 479.747,A -85,B 0,C 180,E1 -1384.116,E2 -1384.116} C_VEL
LIN {X 0,Y 587.271,Z 488.826,A -85,B 0,C 180,E1 -1385.059,E2 -1385.059} C_VEL
LIN {X 0,Y 587.24,Z 496.955,A -85,B 0,C 180,E1 -1386.099,E2 -1386.099} C_VEL
LIN {X 0,Y 587.204,Z 503.757,A -85,B 0,C 180,E1 -1387.186,E2 -1387.186} C_VEL
LIN {X 0,Y 587.185,Z 508.463,A -85,B 0,C 180,E1 -1388.129,E2 -1388.129} C_VEL
LIN {X 0,Y 587.152,Z 513.219,A -85,B 0,C 180,E1 -1389.374,E2 -1389.374} C_VEL
LIN {X 0,Y 587.158,Z 515.724,A -85,B 0,C 180,E1 -1390.267,E2 -1390.267} C_VEL
LIN {X 0,Y 587.121,Z 517.503,A -85,B 0,C 180,E1 -1391.175,E2 -1391.175} C_VEL
LIN {X 0,Y 587.161,Z 518.6,A -85,B 0,C 180,E1 -1392.089,E2 -1392.089} C_VEL
LIN {X 0,Y 587.144,Z 518.994,A -85,B 0,C 180,E1 -1393.1,E2 -1393.1} C_VEL
LIN {X 0,Y 587.152,Z 518.533,A -85,B 0,C 180,E1 -1394.096,E2 -1394.096} C_VEL
LIN {X 0,Y 587.168,Z 517.247,A -85,B 0,C 180,E1 -1395.074,E2 -1395.074} C_VEL
LIN {X 0,Y 587.148,Z 515.183,A -85,B 0,C 180,E1 -1396.033,E2 -1396.033} C_VEL
LIN {X 0,Y 587.178,Z 512.332,A -85,B 0,C 180,E1 -1396.981,E2 -1396.981} C_VEL
LIN {X 0,Y 587.188,Z 507.608,A -85,B 0,C 180,E1 -1398.143,E2 -1398.143} C_VEL
LIN {X 0,Y 587.186,Z 501.227,A -85,B 0,C 180,E1 -1399.338,E2 -1399.338} C_VEL
LIN {X 0,Y 587.263,Z 493.399,A -85,B 0,C 180,E1 -1400.474,E2 -1400.474} C_VEL
LIN {X 0,Y 587.326,Z 484.353,A -85,B 0,C 180,E1 -1401.52,E2 -1401.52} C_VEL
LIN {X 0,Y 587.369,Z 475.007,A -85,B 0,C 180,E1 -1402.394,E2 -1402.394} C_VEL
LIN {X 0,Y 587.416,Z 465.059,A -85,B 0,C 180,E1 -1403.151,E2 -1403.151} C_VEL
LIN {X 0,Y 587.516,Z 454.564,A -85,B 0,C 180,E1 -1403.798,E2 -1403.798} C_VEL
LIN {X 0,Y 587.579,Z 442.923,A -85,B 0,C 180,E1 -1404.366,E2 -1404.366} C_VEL
LIN {X 0,Y 587.641,Z 430.182,A -85,B 0,C 180,E1 -1404.829,E2 -1404.829} C_VEL
LIN {X 0,Y 587.656,Z 418.056,A -85,B 0,C 180,E1 -1405.132,E2 -1405.132} C_VEL
LIN {X 0,Y 587.158,Z 414.919,A -85,B 0,C 180,E1 -1405.208,E2 -1405.208} C_VEL
LIN {X 0,Y 587.141,Z 411.04,A -85,B 0,C 180,E1 -1407.409,E2 -1407.409} C_VEL
LIN {X 0,Y 587.154,Z 406.833,A -85,B 0,C 180,E1 -1409.82,E2 -1409.82} C_VEL
LIN {X 0,Y 587.164,Z 402.49,A -85,B 0,C 180,E1 -1412.341,E2 -1412.341} C_VEL
LIN {X 0,Y 587.177,Z 398.864,A -85,B 0,C 180,E1 -1414.476,E2 -1414.476} C_VEL
LIN {X 0,Y 587.222,Z 393.848,A -85,B 0,C 180,E1 -1417.481,E2 -1417.481} C_VEL
LIN {X 0,Y 587.205,Z 390.238,A -85,B 0,C 180,E1 -1419.691,E2 -1419.691} C_VEL
LIN {X 0,Y 587.229,Z 387.006,A -85,B 0,C 180,E1 -1421.87,E2 -1421.87} C_VEL
LIN {X 0,Y 587.241,Z 383.658,A -85,B 0,C 180,E1 -1424.022,E2 -1424.022} C_VEL
LIN {X 0,Y 587.291,Z 380.396,A -85,B 0,C 180,E1 -1426.153,E2 -1426.153} C_VEL
LIN {X 0,Y 587.29,Z 377.334,A -85,B 0,C 180,E1 -1428.262,E2 -1428.262} C_VEL
LIN {X 0,Y 587.344,Z 377.326,A -85,B 0,C 180,E1 -1431.051,E2 -1431.051} C_VEL
LIN {X 0,Y 587.371,Z 377.323,A -85,B 0,C 180,E1 -1433.265,E2 -1433.265} C_VEL
LIN {X 0,Y 587.31,Z 377.329,A -85,B 0,C 180,E1 -1435.883,E2 -1435.883} C_VEL
LIN {X 0,Y 587.359,Z 377.323,A -85,B 0,C 180,E1 -1437.943,E2 -1437.943} C_VEL
LIN {X 0,Y 587.394,Z 377.321,A -85,B 0,C 180,E1 -1440.686,E2 -1440.686} C_VEL
LIN {X 0,Y 587.331,Z 377.326,A -85,B 0,C 180,E1 -1443.43,E2 -1443.43} C_VEL
LIN {X 0,Y 587.33,Z 377.327,A -85,B 0,C 180,E1 -1446.182,E2 -1446.182} C_VEL
LIN {X 0,Y 587.34,Z 377.327,A -85,B 0,C 180,E1 -1448.949,E2 -1448.949} C_VEL
LIN {X 0,Y 587.34,Z 377.325,A -85,B 0,C 180,E1 -1451.737,E2 -1451.737} C_VEL
LIN {X 0,Y 587.337,Z 377.326,A -85,B 0,C 180,E1 -1454.554,E2 -1454.554} C_VEL
LIN {X 0,Y 587.357,Z 377.326,A -85,B 0,C 180,E1 -1457.406,E2 -1457.406} C_VEL
LIN {X 0,Y 587.332,Z 377.327,A -85,B 0,C 180,E1 -1460.305,E2 -1460.305} C_VEL
LIN {X 0,Y 587.319,Z 377.328,A -85,B 0,C 180,E1 -1463.259,E2 -1463.259} C_VEL
LIN {X 0,Y 587.335,Z 377.327,A -85,B 0,C 180,E1 -1465.517,E2 -1465.517} C_VEL
LIN {X 0,Y 587.346,Z 377.327,A -85,B 0,C 180,E1 -1467.818,E2 -1467.818} C_VEL
LIN {X 0,Y 587.345,Z 377.325,A -85,B 0,C 180,E1 -1470.512,E2 -1470.512} C_VEL
LIN {X 0,Y 587.331,Z 377.327,A -85,B 0,C 180,E1 -1473.397,E2 -1473.397} C_VEL
LIN {X 0,Y 587.345,Z 377.326,A -85,B 0,C 180,E1 -1475.896,E2 -1475.896} C_VEL
LIN {X 0,Y 587.333,Z 377.327,A -85,B 0,C 180,E1 -1478.479,E2 -1478.479} C_VEL
LIN {X 0,Y 587.336,Z 377.328,A -85,B 0,C 180,E1 -1481.157,E2 -1481.157} C_VEL
LIN {X 0,Y 587.325,Z 377.328,A -85,B 0,C 180,E1 -1484.114,E2 -1484.114} C_VEL
LIN {X 0,Y 587.313,Z 377.329,A -85,B 0,C 180,E1 -1486.994,E2 -1486.994} C_VEL
LIN {X 0,Y 587.317,Z 377.33,A -85,B 0,C 180,E1 -1489.747,E2 -1489.747} C_VEL
LIN {X 0,Y 587.346,Z 377.325,A -85,B 0,C 180,E1 -1492.393,E2 -1492.393} C_VEL
LIN {X 0,Y 587.383,Z 377.424,A -85,B 0,C 180,E1 -1493.895,E2 -1493.895} C_VEL
LIN {X 0,Y 587.564,Z 382.607,A -85,B 0,C 180,E1 -1495.794,E2 -1495.794} C_VEL
LIN {X 0,Y 587.489,Z 389.639,A -85,B 0,C 180,E1 -1498.241,E2 -1498.241} C_VEL
LIN {X 0,Y 587.455,Z 397.538,A -85,B 0,C 180,E1 -1500.849,E2 -1500.849} C_VEL
LIN {X 0,Y 587.406,Z 406.675,A -85,B 0,C 180,E1 -1503.81,E2 -1503.81} C_VEL
LIN {X 0,Y 587.331,Z 415.878,A -85,B 0,C 180,E1 -1506.742,E2 -1506.742} C_VEL
LIN {X 0,Y 587.326,Z 424.178,A -85,B 0,C 180,E1 -1509.335,E2 -1509.335} C_VEL
LIN {X 0,Y 587.286,Z 433.628,A -85,B 0,C 180,E1 -1512.233,E2 -1512.233} C_VEL
LIN {X 0,Y 587.219,Z 443.095,A -85,B 0,C 180,E1 -1515.089,E2 -1515.089} C_VEL
LIN {X 0,Y 587.201,Z 452.192,A -85,B 0,C 180,E1 -1517.801,E2 -1517.801} C_VEL
LIN {X 0,Y 587.73,Z 457.248,A -85,B 0,C 180,E1 -1517.899,E2 -1517.899} C_VEL
LIN {X 0,Y 587.682,Z 470.509,A -85,B 0,C 180,E1 -1518.227,E2 -1518.227} C_VEL
LIN {X 0,Y 587.566,Z 482.392,A -85,B 0,C 180,E1 -1518.656,E2 -1518.656} C_VEL
LIN {X 0,Y 587.482,Z 494.217,A -85,B 0,C 180,E1 -1519.227,E2 -1519.227} C_VEL
LIN {X 0,Y 587.468,Z 505.483,A -85,B 0,C 180,E1 -1519.924,E2 -1519.924} C_VEL
LIN {X 0,Y 587.384,Z 515.651,A -85,B 0,C 180,E1 -1520.705,E2 -1520.705} C_VEL
LIN {X 0,Y 587.339,Z 524.79,A -85,B 0,C 180,E1 -1521.571,E2 -1521.571} C_VEL
LIN {X 0,Y 587.258,Z 533.693,A -85,B 0,C 180,E1 -1522.609,E2 -1522.609} C_VEL
LIN {X 0,Y 587.195,Z 540.746,A -85,B 0,C 180,E1 -1523.627,E2 -1523.627} C_VEL
LIN {X 0,Y 587.211,Z 545.682,A -85,B 0,C 180,E1 -1524.506,E2 -1524.506} C_VEL
LIN {X 0,Y 587.188,Z 550.373,A -85,B 0,C 180,E1 -1525.538,E2 -1525.538} C_VEL
LIN {X 0,Y 587.193,Z 553.957,A -85,B 0,C 180,E1 -1526.569,E2 -1526.569} C_VEL
LIN {X 0,Y 587.132,Z 555.809,A -85,B 0,C 180,E1 -1527.256,E2 -1527.256} C_VEL
LIN {X 0,Y 587.141,Z 557.201,A -85,B 0,C 180,E1 -1527.942,E2 -1527.942} C_VEL
LIN {X 0,Y 587.14,Z 558.784,A -85,B 0,C 180,E1 -1529.314,E2 -1529.314} C_VEL
LIN {X 0,Y 587.137,Z 559,A -85,B 0,C 180,E1 -1530,E2 -1530} C_VEL
LIN {X 0,Y 587.147,Z 558.185,A -85,B 0,C 180,E1 -1531.372,E2 -1531.372} C_VEL
LIN {X 0,Y 587.141,Z 557.201,A -85,B 0,C 180,E1 -1532.058,E2 -1532.058} C_VEL
LIN {X 0,Y 587.132,Z 555.809,A -85,B 0,C 180,E1 -1532.745,E2 -1532.745} C_VEL
LIN {X 0,Y 587.213,Z 552.895,A -85,B 0,C 180,E1 -1533.775,E2 -1533.775} C_VEL
LIN {X 0,Y 587.147,Z 548.948,A -85,B 0,C 180,E1 -1534.807,E2 -1534.807} C_VEL
LIN {X 0,Y 587.217,Z 542.876,A -85,B 0,C 180,E1 -1536.011,E2 -1536.011} C_VEL
LIN {X 0,Y 587.245,Z 536.235,A -85,B 0,C 180,E1 -1537.046,E2 -1537.046} C_VEL
LIN {X 0,Y 587.299,Z 527.988,A -85,B 0,C 180,E1 -1538.083,E2 -1538.083} C_VEL
LIN {X 0,Y 587.343,Z 519.535,A -85,B 0,C 180,E1 -1538.949,E2 -1538.949} C_VEL
LIN {X 0,Y 587.421,Z 509.092,A -85,B 0,C 180,E1 -1539.816,E2 -1539.816} C_VEL
LIN {X 0,Y 587.479,Z 498.755,A -85,B 0,C 180,E1 -1540.512,E2 -1540.512} C_VEL
LIN {X 0,Y 587.532,Z 487.139,A -85,B 0,C 180,E1 -1541.134,E2 -1541.134} C_VEL
LIN {X 0,Y 587.623,Z 474.678,A -85,B 0,C 180,E1 -1541.637,E2 -1541.637} C_VEL
LIN {X 0,Y 587.708,Z 461.429,A -85,B 0,C 180,E1 -1542.014,E2 -1542.014} C_VEL
LIN {X 0,Y 587.554,Z 454.484,A -85,B 0,C 180,E1 -1542.157,E2 -1542.157} C_VEL
LIN {X 0,Y 587.2,Z 452.116,A -85,B 0,C 180,E1 -1542.222,E2 -1542.222} C_VEL
LIN {X 0,Y 587.22,Z 443.093,A -85,B 0,C 180,E1 -1544.911,E2 -1544.911} C_VEL
LIN {X 0,Y 587.286,Z 433.626,A -85,B 0,C 180,E1 -1547.768,E2 -1547.768} C_VEL
LIN {X 0,Y 587.326,Z 424.176,A -85,B 0,C 180,E1 -1550.666,E2 -1550.666} C_VEL
LIN {X 0,Y 587.332,Z 415.876,A -85,B 0,C 180,E1 -1553.258,E2 -1553.258} C_VEL
LIN {X 0,Y 587.405,Z 406.41,A -85,B 0,C 180,E1 -1556.275,E2 -1556.275} C_VEL
LIN {X 0,Y 587.464,Z 396.856,A -85,B 0,C 180,E1 -1559.373,E2 -1559.373} C_VEL
LIN {X 0,Y 587.502,Z 388.455,A -85,B 0,C 180,E1 -1562.176,E2 -1562.176} C_VEL
LIN {X 0,Y 587.556,Z 382.154,A -85,B 0,C 180,E1 -1564.377,E2 -1564.377} C_VEL
LIN {X 0,Y 587.457,Z 377.985,A -85,B 0,C 180,E1 -1565.888,E2 -1565.888} C_VEL
LIN {X 0,Y 587.333,Z 377.329,A -85,B 0,C 180,E1 -1566.215,E2 -1566.215} C_VEL
LIN {X 0,Y 587.329,Z 377.328,A -85,B 0,C 180,E1 -1568.941,E2 -1568.941} C_VEL
LIN {X 0,Y 587.355,Z 377.324,A -85,B 0,C 180,E1 -1572.072,E2 -1572.072} C_VEL
LIN {X 0,Y 587.307,Z 377.329,A -85,B 0,C 180,E1 -1575.088,E2 -1575.088} C_VEL
LIN {X 0,Y 587.325,Z 377.327,A -85,B 0,C 180,E1 -1577.925,E2 -1577.925} C_VEL
LIN {X 0,Y 587.325,Z 377.327,A -85,B 0,C 180,E1 -1581.059,E2 -1581.059} C_VEL
LIN {X 0,Y 587.354,Z 377.324,A -85,B 0,C 180,E1 -1583.292,E2 -1583.292} C_VEL
LIN {X 0,Y 587.335,Z 377.325,A -85,B 0,C 180,E1 -1585.778,E2 -1585.778} C_VEL
LIN {X 0,Y 587.342,Z 377.324,A -85,B 0,C 180,E1 -1588.231,E2 -1588.231} C_VEL
LIN {X 0,Y 587.351,Z 377.323,A -85,B 0,C 180,E1 -1590.866,E2 -1590.866} C_VEL
LIN {X 0,Y 587.356,Z 377.325,A -85,B 0,C 180,E1 -1593.819,E2 -1593.819} C_VEL
LIN {X 0,Y 587.337,Z 377.326,A -85,B 0,C 180,E1 -1595.993,E2 -1595.993} C_VEL
LIN {X 0,Y 587.322,Z 377.327,A -85,B 0,C 180,E1 -1598.226,E2 -1598.226} C_VEL
LIN {X 0,Y 587.349,Z 377.325,A -85,B 0,C 180,E1 -1601.151,E2 -1601.151} C_VEL
LIN {X 0,Y 587.348,Z 377.327,A -85,B 0,C 180,E1 -1603.311,E2 -1603.311} C_VEL
LIN {X 0,Y 587.357,Z 377.322,A -85,B 0,C 180,E1 -1606.154,E2 -1606.154} C_VEL
LIN {X 0,Y 587.343,Z 377.325,A -85,B 0,C 180,E1 -1608.962,E2 -1608.962} C_VEL
LIN {X 0,Y 587.366,Z 377.324,A -85,B 0,C 180,E1 -1611.745,E2 -1611.745} C_VEL
LIN {X 0,Y 587.357,Z 377.323,A -85,B 0,C 180,E1 -1614.507,E2 -1614.507} C_VEL
LIN {X 0,Y 587.378,Z 377.32,A -85,B 0,C 180,E1 -1617.257,E2 -1617.257} C_VEL
LIN {X 0,Y 587.383,Z 377.322,A -85,B 0,C 180,E1 -1620,E2 -1620} C_VEL
LIN {X 0,Y 587.38,Z 377.32,A -85,B 0,C 180,E1 -1622.743,E2 -1622.743} C_VEL
LIN {X 0,Y 587.355,Z 377.322,A -85,B 0,C 180,E1 -1625.493,E2 -1625.493} C_VEL
LIN {X 0,Y 587.366,Z 377.323,A -85,B 0,C 180,E1 -1628.255,E2 -1628.255} C_VEL
LIN {X 0,Y 587.348,Z 377.324,A -85,B 0,C 180,E1 -1631.134,E2 -1631.134} C_VEL
LIN {X 0,Y 587.365,Z 377.324,A -85,B 0,C 180,E1 -1634.26,E2 -1634.26} C_VEL
LIN {X 0,Y 587.356,Z 377.322,A -85,B 0,C 180,E1 -1637.406,E2 -1637.406} C_VEL
LIN {X 0,Y 587.323,Z 377.327,A -85,B 0,C 180,E1 -1638.309,E2 -1638.309} C_VEL
LIN {X 0,Y 586.67,Z 377.41,A -85,B 0,C 180,E1 -1638.881,E2 -1638.881} C_VEL
LIN {X 0,Y 583.84,Z 377.764,A -85,B 0,C 180,E1 -1639.809,E2 -1639.809} C_VEL
LIN {X 0,Y 581.431,Z 378.066,A -85,B 0,C 180,E1 -1640.556,E2 -1640.556} C_VEL
LIN {X 0,Y 580.378,Z 378.195,A -85,B 0,C 180,E1 -1641.132,E2 -1641.132} C_VEL
LIN {X 0,Y 580.282,Z 378.205,A -85,B 0,C 180,E1 -1641.327,E2 -1641.327} C_VEL
LIN {X 0,Y 580.28,Z 378.204,A -85,B 0,C 180,E1 -1643.558,E2 -1643.558} C_VEL
LIN {X 0,Y 580.278,Z 378.204,A -85,B 0,C 180,E1 -1645.85,E2 -1645.85} C_VEL
LIN {X 0,Y 580.297,Z 378.202,A -85,B 0,C 180,E1 -1648.186,E2 -1648.186} C_VEL
LIN {X 0,Y 580.285,Z 378.204,A -85,B 0,C 180,E1 -1650.695,E2 -1650.695} C_VEL
LIN {X 0,Y 580.306,Z 378.203,A -85,B 0,C 180,E1 -1653.317,E2 -1653.317} C_VEL
LIN {X 0,Y 580.295,Z 378.202,A -85,B 0,C 180,E1 -1656.402,E2 -1656.402} C_VEL
LIN {X 0,Y 580.297,Z 378.203,A -85,B 0,C 180,E1 -1659.185,E2 -1659.185} C_VEL
LIN {X 0,Y 580.289,Z 378.206,A -85,B 0,C 180,E1 -1661.768,E2 -1661.768} C_VEL
LIN {X 0,Y 580.262,Z 378.206,A -85,B 0,C 180,E1 -1664.627,E2 -1664.627} C_VEL
LIN {X 0,Y 580.287,Z 378.205,A -85,B 0,C 180,E1 -1667.628,E2 -1667.628} C_VEL
LIN {X 0,Y 580.286,Z 378.205,A -85,B 0,C 180,E1 -1670.067,E2 -1670.067} C_VEL
LIN {X 0,Y 580.302,Z 378.201,A -85,B 0,C 180,E1 -1673.066,E2 -1673.066} C_VEL
LIN {X 0,Y 580.316,Z 378.203,A -85,B 0,C 180,E1 -1676.145,E2 -1676.145} C_VEL
LIN {X 0,Y 580.277,Z 378.207,A -85,B 0,C 180,E1 -1678.615,E2 -1678.615} C_VEL
LIN {X 0,Y 580.292,Z 378.204,A -85,B 0,C 180,E1 -1681.024,E2 -1681.024} C_VEL
LIN {X 0,Y 580.295,Z 378.202,A -85,B 0,C 180,E1 -1683.666,E2 -1683.666} C_VEL
LIN {X 0,Y 580.303,Z 378.204,A -85,B 0,C 180,E1 -1685.684,E2 -1685.684} C_VEL
LIN {X 0,Y 580.269,Z 378.207,A -85,B 0,C 180,E1 -1687.947,E2 -1687.947} C_VEL
LIN {X 0,Y 580.301,Z 378.201,A -85,B 0,C 180,E1 -1690.913,E2 -1690.913} C_VEL
LIN {X 0,Y 580.268,Z 378.207,A -85,B 0,C 180,E1 -1693.825,E2 -1693.825} C_VEL
LIN {X 0,Y 580.328,Z 378.198,A -85,B 0,C 180,E1 -1695.983,E2 -1695.983} C_VEL
LIN {X 0,Y 580.308,Z 378.203,A -85,B 0,C 180,E1 -1698.827,E2 -1698.827} C_VEL
LIN {X 0,Y 580.331,Z 378.197,A -85,B 0,C 180,E1 -1701.644,E2 -1701.644} C_VEL
LIN {X 0,Y 580.331,Z 378.198,A -85,B 0,C 180,E1 -1704.44,E2 -1704.44} C_VEL
LIN {X 0,Y 580.346,Z 378.196,A -85,B 0,C 180,E1 -1707.918,E2 -1707.918} C_VEL
LIN {X 0,Y 580.366,Z 378.197,A -85,B 0,C 180,E1 -1710.694,E2 -1710.694} C_VEL
LIN {X 0,Y 580.288,Z 378.203,A -85,B 0,C 180,E1 -1713.471,E2 -1713.471} C_VEL
LIN {X 0,Y 580.324,Z 378.201,A -85,B 0,C 180,E1 -1715.559,E2 -1715.559} C_VEL
LIN {X 0,Y 580.248,Z 378.209,A -85,B 0,C 180,E1 -1717.656,E2 -1717.656} C_VEL
LIN {X 0,Y 580.213,Z 378.626,A -85,B 0,C 180,E1 -1718.357,E2 -1718.357} C_VEL
LIN {X 0,Y 580.225,Z 382.86,A -85,B 0,C 180,E1 -1721.174,E2 -1721.174} C_VEL
LIN {X 0,Y 580.198,Z 387.688,A -85,B 0,C 180,E1 -1724.292,E2 -1724.292} C_VEL
LIN {X 0,Y 580.105,Z 391.673,A -85,B 0,C 180,E1 -1726.903,E2 -1726.903} C_VEL
LIN {X 0,Y 580.071,Z 396.37,A -85,B 0,C 180,E1 -1729.83,E2 -1729.83} C_VEL
LIN {X 0,Y 580.044,Z 401.56,A -85,B 0,C 180,E1 -1732.95,E2 -1732.95} C_VEL
LIN {X 0,Y 580.064,Z 405.179,A -85,B 0,C 180,E1 -1735.09,E2 -1735.09} C_VEL
LIN {X 0,Y 580.025,Z 409.839,A -85,B 0,C 180,E1 -1737.807,E2 -1737.807} C_VEL
LIN {X 0,Y 580.033,Z 414.905,A -85,B 0,C 180,E1 -1740.722,E2 -1740.722} C_VEL
LIN {X 0,Y 580.785,Z 421.113,A -85,B 0,C 180,E1 -1740.878,E2 -1740.878} C_VEL
LIN {X 0,Y 580.677,Z 434.477,A -85,B 0,C 180,E1 -1741.26,E2 -1741.26} C_VEL
LIN {X 0,Y 580.535,Z 447.174,A -85,B 0,C 180,E1 -1741.776,E2 -1741.776} C_VEL
LIN {X 0,Y 580.397,Z 458.682,A -85,B 0,C 180,E1 -1742.399,E2 -1742.399} C_VEL
LIN {X 0,Y 580.391,Z 469.975,A -85,B 0,C 180,E1 -1743.175,E2 -1743.175} C_VEL
LIN {X 0,Y 580.314,Z 480.333,A -85,B 0,C 180,E1 -1744.063,E2 -1744.063} C_VEL
LIN {X 0,Y 580.234,Z 488.396,A -85,B 0,C 180,E1 -1744.911,E2 -1744.911} C_VEL
LIN {X 0,Y 580.182,Z 495.937,A -85,B 0,C 180,E1 -1745.87,E2 -1745.87} C_VEL
LIN {X 0,Y 580.131,Z 503.512,A -85,B 0,C 180,E1 -1747.07,E2 -1747.07} C_VEL
LIN {X 0,Y 580.097,Z 508.868,A -85,B 0,C 180,E1 -1748.161,E2 -1748.161} C_VEL
LIN {X 0,Y 580.07,Z 512.676,A -85,B 0,C 180,E1 -1749.158,E2 -1749.158} C_VEL
LIN {X 0,Y 580.059,Z 515.751,A -85,B 0,C 180,E1 -1750.243,E2 -1750.243} C_VEL
LIN {X 0,Y 580.034,Z 517.744,A -85,B 0,C 180,E1 -1751.303,E2 -1751.303} C_VEL
LIN {X 0,Y 580.054,Z 518.935,A -85,B 0,C 180,E1 -1752.726,E2 -1752.726} C_VEL
LIN {X 0,Y 580.023,Z 518.823,A -85,B 0,C 180,E1 -1753.681,E2 -1753.681} C_VEL
LIN {X 0,Y 580.065,Z 517.943,A -85,B 0,C 180,E1 -1754.645,E2 -1754.645} C_VEL
LIN {X 0,Y 580.073,Z 516.225,A -85,B 0,C 180,E1 -1755.628,E2 -1755.628} C_VEL
LIN {X 0,Y 580.057,Z 513.612,A -85,B 0,C 180,E1 -1756.632,E2 -1756.632} C_VEL
LIN {X 0,Y 580.111,Z 508.849,A -85,B 0,C 180,E1 -1757.934,E2 -1757.934} C_VEL
LIN {X 0,Y 580.111,Z 502.817,A -85,B 0,C 180,E1 -1759.14,E2 -1759.14} C_VEL
LIN {X 0,Y 580.176,Z 495.634,A -85,B 0,C 180,E1 -1760.263,E2 -1760.263} C_VEL
LIN {X 0,Y 580.242,Z 488.346,A -85,B 0,C 180,E1 -1761.185,E2 -1761.185} C_VEL
LIN {X 0,Y 580.287,Z 479.465,A -85,B 0,C 180,E1 -1762.11,E2 -1762.11} C_VEL
LIN {X 0,Y 580.411,Z 469.805,A -85,B 0,C 180,E1 -1762.927,E2 -1762.927} C_VEL
LIN {X 0,Y 580.489,Z 458.602,A -85,B 0,C 180,E1 -1763.694,E2 -1763.694} C_VEL
LIN {X 0,Y 580.596,Z 446.952,A -85,B 0,C 180,E1 -1764.323,E2 -1764.323} C_VEL
LIN {X 0,Y 580.676,Z 435.31,A -85,B 0,C 180,E1 -1764.801,E2 -1764.801} C_VEL
LIN {X 0,Y 580.779,Z 421.95,A -85,B 0,C 180,E1 -1765.192,E2 -1765.192} C_VEL
LIN {X 0,Y 580.493,Z 417.638,A -85,B 0,C 180,E1 -1765.291,E2 -1765.291} C_VEL
LIN {X 0,Y 580.069,Z 414.912,A -85,B 0,C 180,E1 -1765.363,E2 -1765.363} C_VEL
LIN {X 0,Y 580.045,Z 410.312,A -85,B 0,C 180,E1 -1768.009,E2 -1768.009} C_VEL
LIN {X 0,Y 580.079,Z 405.64,A -85,B 0,C 180,E1 -1770.728,E2 -1770.728} C_VEL
LIN {X 0,Y 580.121,Z 400.618,A -85,B 0,C 180,E1 -1773.699,E2 -1773.699} C_VEL
LIN {X 0,Y 580.116,Z 396.079,A -85,B 0,C 180,E1 -1776.435,E2 -1776.435} C_VEL
LIN {X 0,Y 580.158,Z 391.33,A -85,B 0,C 180,E1 -1779.433,E2 -1779.433} C_VEL
LIN {X 0,Y 580.165,Z 388.106,A -85,B 0,C 180,E1 -1781.642,E2 -1781.642} C_VEL
LIN {X 0,Y 580.203,Z 384.689,A -85,B 0,C 180,E1 -1783.823,E2 -1783.823} C_VEL
LIN {X 0,Y 580.235,Z 381.393,A -85,B 0,C 180,E1 -1785.981,E2 -1785.981} C_VEL
LIN {X 0,Y 580.22,Z 378.215,A -85,B 0,C 180,E1 -1788.117,E2 -1788.117} C_VEL
LIN {X 0,Y 580.275,Z 378.208,A -85,B 0,C 180,E1 -1790.238,E2 -1790.238} C_VEL
LIN {X 0,Y 580.33,Z 378.201,A -85,B 0,C 180,E1 -1792.345,E2 -1792.345} C_VEL
LIN {X 0,Y 580.338,Z 378.198,A -85,B 0,C 180,E1 -1795.137,E2 -1795.137} C_VEL
LIN {X 0,Y 580.33,Z 378.199,A -85,B 0,C 180,E1 -1797.918,E2 -1797.918} C_VEL
LIN {X 0,Y 580.364,Z 378.197,A -85,B 0,C 180,E1 -1800.694,E2 -1800.694} C_VEL
LIN {X 0,Y 580.283,Z 378.205,A -85,B 0,C 180,E1 -1803.472,E2 -1803.472} C_VEL
LIN {X 0,Y 580.323,Z 378.2,A -85,B 0,C 180,E1 -1805.56,E2 -1805.56} C_VEL
LIN {X 0,Y 580.331,Z 378.199,A -85,B 0,C 180,E1 -1808.356,E2 -1808.356} C_VEL
LIN {X 0,Y 580.295,Z 378.205,A -85,B 0,C 180,E1 -1811.191,E2 -1811.191} C_VEL
LIN {X 0,Y 580.324,Z 378.2,A -85,B 0,C 180,E1 -1814.017,E2 -1814.017} C_VEL
LIN {X 0,Y 580.313,Z 378.201,A -85,B 0,C 180,E1 -1816.916,E2 -1816.916} C_VEL
LIN {X 0,Y 580.305,Z 378.202,A -85,B 0,C 180,E1 -1819.822,E2 -1819.822} C_VEL
LIN {X 0,Y 580.272,Z 378.206,A -85,B 0,C 180,E1 -1822.053,E2 -1822.053} C_VEL
LIN {X 0,Y 580.305,Z 378.202,A -85,B 0,C 180,E1 -1825.08,E2 -1825.08} C_VEL
LIN {X 0,Y 580.317,Z 378.202,A -85,B 0,C 180,E1 -1827.863,E2 -1827.863} C_VEL
LIN {X 0,Y 580.292,Z 378.204,A -85,B 0,C 180,E1 -1830.697,E2 -1830.697} C_VEL
LIN {X 0,Y 580.3,Z 378.203,A -85,B 0,C 180,E1 -1833.317,E2 -1833.317} C_VEL
LIN {X 0,Y 580.311,Z 378.201,A -85,B 0,C 180,E1 -1835.766,E2 -1835.766} C_VEL
LIN {X 0,Y 580.288,Z 378.207,A -85,B 0,C 180,E1 -1838.147,E2 -1838.147} C_VEL
LIN {X 0,Y 580.299,Z 378.203,A -85,B 0,C 180,E1 -1840.844,E2 -1840.844} C_VEL
LIN {X 0,Y 580.277,Z 378.206,A -85,B 0,C 180,E1 -1843.658,E2 -1843.658} C_VEL
LIN {X 0,Y 580.272,Z 378.207,A -85,B 0,C 180,E1 -1846.61,E2 -1846.61} C_VEL
LIN {X 0,Y 580.298,Z 378.203,A -85,B 0,C 180,E1 -1849.157,E2 -1849.157} C_VEL
LIN {X 0,Y 580.29,Z 378.205,A -85,B 0,C 180,E1 -1851.927,E2 -1851.927} C_VEL
LIN {X 0,Y 580.346,Z 378.24,A -85,B 0,C 180,E1 -1853.694,E2 -1853.694} C_VEL
LIN {X 0,Y 580.594,Z 382.825,A -85,B 0,C 180,E1 -1855.4,E2 -1855.4} C_VEL
LIN {X 0,Y 580.493,Z 389.941,A -85,B 0,C 180,E1 -1857.94,E2 -1857.94} C_VEL
LIN {X 0,Y 580.464,Z 398.062,A -85,B 0,C 180,E1 -1860.662,E2 -1860.662} C_VEL
LIN {X 0,Y 580.378,Z 407.221,A -85,B 0,C 180,E1 -1863.649,E2 -1863.649} C_VEL
LIN {X 0,Y 580.302,Z 415.878,A -85,B 0,C 180,E1 -1866.444,E2 -1866.444} C_VEL
LIN {X 0,Y 580.266,Z 423.455,A -85,B 0,C 180,E1 -1868.844,E2 -1868.844} C_VEL
LIN {X 0,Y 580.224,Z 432.445,A -85,B 0,C 180,E1 -1871.644,E2 -1871.644} C_VEL
LIN {X 0,Y 580.183,Z 440.728,A -85,B 0,C 180,E1 -1874.184,E2 -1874.184} C_VEL
LIN {X 0,Y 580.136,Z 450.195,A -85,B 0,C 180,E1 -1877.049,E2 -1877.049} C_VEL
LIN {X 0,Y 580.123,Z 452.192,A -85,B 0,C 180,E1 -1877.649,E2 -1877.649} C_VEL
LIN {X 0,Y 580.804,Z 457.248,A -85,B 0,C 180,E1 -1877.753,E2 -1877.753} C_VEL
LIN {X 0,Y 580.715,Z 470.51,A -85,B 0,C 180,E1 -1878.083,E2 -1878.083} C_VEL
LIN {X 0,Y 580.61,Z 482.327,A -85,B 0,C 180,E1 -1878.515,E2 -1878.515} C_VEL
LIN {X 0,Y 580.497,Z 494.218,A -85,B 0,C 180,E1 -1879.096,E2 -1879.096} C_VEL
LIN {X 0,Y 580.458,Z 505.484,A -85,B 0,C 180,E1 -1879.801,E2 -1879.801} C_VEL
LIN {X 0,Y 580.352,Z 515.651,A -85,B 0,C 180,E1 -1880.591,E2 -1880.591} C_VEL
LIN {X 0,Y 580.279,Z 524.79,A -85,B 0,C 180,E1 -1881.468,E2 -1881.468} C_VEL
LIN {X 0,Y 580.199,Z 533.693,A -85,B 0,C 180,E1 -1882.518,E2 -1882.518} C_VEL
LIN {X 0,Y 580.11,Z 541.282,A -85,B 0,C 180,E1 -1883.639,E2 -1883.639} C_VEL
LIN {X 0,Y 580.086,Z 547.367,A -85,B 0,C 180,E1 -1884.787,E2 -1884.787} C_VEL
LIN {X 0,Y 580.105,Z 551.678,A -85,B 0,C 180,E1 -1885.832,E2 -1885.832} C_VEL
LIN {X 0,Y 580.123,Z 553.958,A -85,B 0,C 180,E1 -1886.528,E2 -1886.528} C_VEL
LIN {X 0,Y 580.043,Z 555.809,A -85,B 0,C 180,E1 -1887.222,E2 -1887.222} C_VEL
LIN {X 0,Y 580.04,Z 557.2,A -85,B 0,C 180,E1 -1887.917,E2 -1887.917} C_VEL
LIN {X 0,Y 580.04,Z 558.785,A -85,B 0,C 180,E1 -1889.306,E2 -1889.306} C_VEL
LIN {X 0,Y 580.037,Z 559,A -85,B 0,C 180,E1 -1890,E2 -1890} C_VEL
LIN {X 0,Y 580.046,Z 558.185,A -85,B 0,C 180,E1 -1891.389,E2 -1891.389} C_VEL
LIN {X 0,Y 580.04,Z 557.2,A -85,B 0,C 180,E1 -1892.083,E2 -1892.083} C_VEL
LIN {X 0,Y 580.043,Z 555.809,A -85,B 0,C 180,E1 -1892.778,E2 -1892.778} C_VEL
LIN {X 0,Y 580.11,Z 552.895,A -85,B 0,C 180,E1 -1893.821,E2 -1893.821} C_VEL
LIN {X 0,Y 580.053,Z 548.948,A -85,B 0,C 180,E1 -1894.865,E2 -1894.865} C_VEL
LIN {X 0,Y 580.139,Z 542.876,A -85,B 0,C 180,E1 -1896.085,E2 -1896.085} C_VEL
LIN {X 0,Y 580.184,Z 536.235,A -85,B 0,C 180,E1 -1897.133,E2 -1897.133} C_VEL
LIN {X 0,Y 580.25,Z 527.988,A -85,B 0,C 180,E1 -1898.182,E2 -1898.182} C_VEL
LIN {X 0,Y 580.308,Z 519.536,A -85,B 0,C 180,E1 -1899.059,E2 -1899.059} C_VEL
LIN {X 0,Y 580.423,Z 509.093,A -85,B 0,C 180,E1 -1899.936,E2 -1899.936} C_VEL
LIN {X 0,Y 580.499,Z 498.754,A -85,B 0,C 180,E1 -1900.64,E2 -1900.64} C_VEL
LIN {X 0,Y 580.564,Z 487.587,A -85,B 0,C 180,E1 -1901.248,E2 -1901.248} C_VEL
LIN {X 0,Y 580.665,Z 475.762,A -85,B 0,C 180,E1 -1901.741,E2 -1901.741} C_VEL
LIN {X 0,Y 580.762,Z 462.342,A -85,B 0,C 180,E1 -1902.138,E2 -1902.138} C_VEL
LIN {X 0,Y 580.577,Z 454.938,A -85,B 0,C 180,E1 -1902.297,E2 -1902.297} C_VEL
LIN {X 0,Y 580.126,Z 452.116,A -85,B 0,C 180,E1 -1902.373,E2 -1902.373} C_VEL
LIN {X 0,Y 580.157,Z 443.093,A -85,B 0,C 180,E1 -1905.097,E2 -1905.097} C_VEL
LIN {X 0,Y 580.209,Z 434.81,A -85,B 0,C 180,E1 -1907.627,E2 -1907.627} C_VEL
LIN {X 0,Y 580.269,Z 425.343,A -85,B 0,C 180,E1 -1910.563,E2 -1910.563} C_VEL
LIN {X 0,Y 580.276,Z 417.611,A -85,B 0,C 180,E1 -1913.004,E2 -1913.004} C_VEL
LIN {X 0,Y 580.367,Z 408.776,A -85,B 0,C 180,E1 -1915.846,E2 -1915.846} C_VEL
LIN {X 0,Y 580.383,Z 400.384,A -85,B 0,C 180,E1 -1918.575,E2 -1918.575} C_VEL
LIN {X 0,Y 580.424,Z 393.922,A -85,B 0,C 180,E1 -1920.717,E2 -1920.717} C_VEL
LIN {X 0,Y 580.557,Z 386.299,A -85,B 0,C 180,E1 -1923.354,E2 -1923.354} C_VEL
LIN {X 0,Y 580.516,Z 379.584,A -85,B 0,C 180,E1 -1925.793,E2 -1925.793} C_VEL
LIN {X 0,Y 580.28,Z 378.207,A -85,B 0,C 180,E1 -1926.403,E2 -1926.403} C_VEL
LIN {X 0,Y 580.306,Z 378.201,A -85,B 0,C 180,E1 -1929.186,E2 -1929.186} C_VEL
LIN {X 0,Y 580.301,Z 378.201,A -85,B 0,C 180,E1 -1931.767,E2 -1931.767} C_VEL
LIN {X 0,Y 580.256,Z 378.21,A -85,B 0,C 180,E1 -1934.627,E2 -1934.627} C_VEL
LIN {X 0,Y 580.279,Z 378.206,A -85,B 0,C 180,E1 -1937.294,E2 -1937.294} C_VEL
LIN {X 0,Y 580.282,Z 378.203,A -85,B 0,C 180,E1 -1940.066,E2 -1940.066} C_VEL
LIN {X 0,Y 580.302,Z 378.205,A -85,B 0,C 180,E1 -1943.065,E2 -1943.065} C_VEL
LIN {X 0,Y 580.3,Z 378.201,A -85,B 0,C 180,E1 -1946.144,E2 -1946.144} C_VEL
LIN {X 0,Y 580.277,Z 378.204,A -85,B 0,C 180,E1 -1948.614,E2 -1948.614} C_VEL
LIN {X 0,Y 580.294,Z 378.203,A -85,B 0,C 180,E1 -1951.024,E2 -1951.024} C_VEL
LIN {X 0,Y 580.29,Z 378.205,A -85,B 0,C 180,E1 -1953.666,E2 -1953.666} C_VEL
LIN {X 0,Y 580.301,Z 378.201,A -85,B 0,C 180,E1 -1955.684,E2 -1955.684} C_VEL
LIN {X 0,Y 580.272,Z 378.204,A -85,B 0,C 180,E1 -1957.947,E2 -1957.947} C_VEL
LIN {X 0,Y 580.299,Z 378.205,A -85,B 0,C 180,E1 -1960.913,E2 -1960.913} C_VEL
LIN {X 0,Y 580.275,Z 378.204,A -85,B 0,C 180,E1 -1963.825,E2 -1963.825} C_VEL
LIN {X 0,Y 580.325,Z 378.199,A -85,B 0,C 180,E1 -1965.983,E2 -1965.983} C_VEL
LIN {X 0,Y 580.305,Z 378.201,A -85,B 0,C 180,E1 -1968.827,E2 -1968.827} C_VEL
LIN {X 0,Y 580.332,Z 378.201,A -85,B 0,C 180,E1 -1971.644,E2 -1971.644} C_VEL
LIN {X 0,Y 580.324,Z 378.199,A -85,B 0,C 180,E1 -1974.44,E2 -1974.44} C_VEL
LIN {X 0,Y 580.344,Z 378.196,A -85,B 0,C 180,E1 -1977.223,E2 -1977.223} C_VEL
LIN {X 0,Y 580.353,Z 378.198,A -85,B 0,C 180,E1 -1980,E2 -1980} C_VEL
LIN {X 0,Y 580.345,Z 378.196,A -85,B 0,C 180,E1 -1982.776,E2 -1982.776} C_VEL
LIN {X 0,Y 580.322,Z 378.199,A -85,B 0,C 180,E1 -1985.56,E2 -1985.56} C_VEL
LIN {X 0,Y 580.332,Z 378.2,A -85,B 0,C 180,E1 -1988.356,E2 -1988.356} C_VEL
LIN {X 0,Y 580.3,Z 378.202,A -85,B 0,C 180,E1 -1991.191,E2 -1991.191} C_VEL
LIN {X 0,Y 580.325,Z 378.198,A -85,B 0,C 180,E1 -1994.017,E2 -1994.017} C_VEL
LIN {X 0,Y 580.312,Z 378.202,A -85,B 0,C 180,E1 -1996.914,E2 -1996.914} C_VEL
LIN {X 0,Y 580.289,Z 378.202,A -85,B 0,C 180,E1 -1999.823,E2 -1999.823} C_VEL
LIN {X 0,Y 580.282,Z 378.205,A -85,B 0,C 180,E1 -2001.327,E2 -2001.327} C_VEL
LIN {X 0,Y 579.584,Z 378.291,A -85,B 0,C 180,E1 -2001.906,E2 -2001.906} C_VEL
LIN {X 0,Y 576.708,Z 378.651,A -85,B 0,C 180,E1 -2002.846,E2 -2002.846} C_VEL
LIN {X 0,Y 574.315,Z 378.948,A -85,B 0,C 180,E1 -2003.603,E2 -2003.603} C_VEL
LIN {X 0,Y 573.317,Z 379.072,A -85,B 0,C 180,E1 -2004.187,E2 -2004.187} C_VEL
LIN {X 0,Y 573.25,Z 379.079,A -85,B 0,C 180,E1 -2004.384,E2 -2004.384} C_VEL
LIN {X 0,Y 573.25,Z 379.08,A -85,B 0,C 180,E1 -2006.976,E2 -2006.976} C_VEL
LIN {X 0,Y 573.245,Z 379.081,A -85,B 0,C 180,E1 -2009.488,E2 -2009.488} C_VEL
LIN {X 0,Y 573.256,Z 379.079,A -85,B 0,C 180,E1 -2012.645,E2 -2012.645} C_VEL
LIN {X 0,Y 573.254,Z 379.079,A -85,B 0,C 180,E1 -2015.185,E2 -2015.185} C_VEL
LIN {X 0,Y 573.237,Z 379.081,A -85,B 0,C 180,E1 -2017.808,E2 -2017.808} C_VEL
LIN {X 0,Y 573.245,Z 379.083,A -85,B 0,C 180,E1 -2020.525,E2 -2020.525} C_VEL
LIN {X 0,Y 573.241,Z 379.081,A -85,B 0,C 180,E1 -2023.359,E2 -2023.359} C_VEL
LIN {X 0,Y 573.239,Z 379.082,A -85,B 0,C 180,E1 -2026.332,E2 -2026.332} C_VEL
LIN {X 0,Y 573.246,Z 379.08,A -85,B 0,C 180,E1 -2028.544,E2 -2028.544} C_VEL
LIN {X 0,Y 573.24,Z 379.084,A -85,B 0,C 180,E1 -2031.298,E2 -2031.298} C_VEL
LIN {X 0,Y 573.246,Z 379.081,A -85,B 0,C 180,E1 -2034.014,E2 -2034.014} C_VEL
LIN {X 0,Y 573.271,Z 379.077,A -85,B 0,C 180,E1 -2036.518,E2 -2036.518} C_VEL
LIN {X 0,Y 573.229,Z 379.082,A -85,B 0,C 180,E1 -2039.118,E2 -2039.118} C_VEL
LIN {X 0,Y 573.235,Z 379.081,A -85,B 0,C 180,E1 -2041.435,E2 -2041.435} C_VEL
LIN {X 0,Y 573.268,Z 379.077,A -85,B 0,C 180,E1 -2043.81,E2 -2043.81} C_VEL
LIN {X 0,Y 573.235,Z 379.082,A -85,B 0,C 180,E1 -2046.135,E2 -2046.135} C_VEL
LIN {X 0,Y 573.252,Z 379.082,A -85,B 0,C 180,E1 -2049.174,E2 -2049.174} C_VEL
LIN {X 0,Y 573.224,Z 379.084,A -85,B 0,C 180,E1 -2051.411,E2 -2051.411} C_VEL
LIN {X 0,Y 573.243,Z 379.08,A -85,B 0,C 180,E1 -2053.621,E2 -2053.621} C_VEL
LIN {X 0,Y 573.276,Z 379.076,A -85,B 0,C 180,E1 -2055.807,E2 -2055.807} C_VEL
LIN {X 0,Y 573.266,Z 379.081,A -85,B 0,C 180,E1 -2058.745,E2 -2058.745} C_VEL
LIN {X 0,Y 573.286,Z 379.075,A -85,B 0,C 180,E1 -2061.54,E2 -2061.54} C_VEL
LIN {X 0,Y 573.298,Z 379.074,A -85,B 0,C 180,E1 -2064.372,E2 -2064.372} C_VEL
LIN {X 0,Y 573.316,Z 379.071,A -85,B 0,C 180,E1 -2067.892,E2 -2067.892} C_VEL
LIN {X 0,Y 573.336,Z 379.072,A -85,B 0,C 180,E1 -2070.702,E2 -2070.702} C_VEL
LIN {X 0,Y 573.239,Z 379.081,A -85,B 0,C 180,E1 -2073.514,E2 -2073.514} C_VEL
LIN {X 0,Y 573.292,Z 379.077,A -85,B 0,C 180,E1 -2075.628,E2 -2075.628} C_VEL
LIN {X 0,Y 573.199,Z 379.088,A -85,B 0,C 180,E1 -2077.751,E2 -2077.751} C_VEL
LIN {X 0,Y 573.168,Z 379.536,A -85,B 0,C 180,E1 -2078.461,E2 -2078.461} C_VEL
LIN {X 0,Y 573.158,Z 383.791,A -85,B 0,C 180,E1 -2081.314,E2 -2081.314} C_VEL
LIN {X 0,Y 573.13,Z 388.452,A -85,B 0,C 180,E1 -2084.364,E2 -2084.364} C_VEL
LIN {X 0,Y 573.041,Z 392.671,A -85,B 0,C 180,E1 -2087.118,E2 -2087.118} C_VEL
LIN {X 0,Y 572.982,Z 397.28,A -85,B 0,C 180,E1 -2090.086,E2 -2090.086} C_VEL
LIN {X 0,Y 572.962,Z 402.257,A -85,B 0,C 180,E1 -2093.111,E2 -2093.111} C_VEL
LIN {X 0,Y 572.967,Z 406.126,A -85,B 0,C 180,E1 -2095.423,E2 -2095.423} C_VEL
LIN {X 0,Y 572.919,Z 410.441,A -85,B 0,C 180,E1 -2097.966,E2 -2097.966} C_VEL
LIN {X 0,Y 572.96,Z 415.027,A -85,B 0,C 180,E1 -2100.584,E2 -2100.584} C_VEL
LIN {X 0,Y 573.832,Z 422.052,A -85,B 0,C 180,E1 -2100.751,E2 -2100.751} C_VEL
LIN {X 0,Y 573.719,Z 434.875,A -85,B 0,C 180,E1 -2101.129,E2 -2101.129} C_VEL
LIN {X 0,Y 573.581,Z 446.874,A -85,B 0,C 180,E1 -2101.624,E2 -2101.624} C_VEL
LIN {X 0,Y 573.415,Z 458.457,A -85,B 0,C 180,E1 -2102.254,E2 -2102.254} C_VEL
LIN {X 0,Y 573.373,Z 469.997,A -85,B 0,C 180,E1 -2103.055,E2 -2103.055} C_VEL
LIN {X 0,Y 573.267,Z 479.842,A -85,B 0,C 180,E1 -2103.903,E2 -2103.903} C_VEL
LIN {X 0,Y 573.174,Z 487.997,A -85,B 0,C 180,E1 -2104.762,E2 -2104.762} C_VEL
LIN {X 0,Y 573.109,Z 495.876,A -85,B 0,C 180,E1 -2105.772,E2 -2105.772} C_VEL
LIN {X 0,Y 573.036,Z 503.182,A -85,B 0,C 180,E1 -2106.938,E2 -2106.938} C_VEL
LIN {X 0,Y 573.001,Z 507.631,A -85,B 0,C 180,E1 -2107.825,E2 -2107.825} C_VEL
LIN {X 0,Y 573.012,Z 512.486,A -85,B 0,C 180,E1 -2109.055,E2 -2109.055} C_VEL
LIN {X 0,Y 572.975,Z 515.371,A -85,B 0,C 180,E1 -2110.057,E2 -2110.057} C_VEL
LIN {X 0,Y 572.946,Z 518.007,A -85,B 0,C 180,E1 -2111.481,E2 -2111.481} C_VEL
LIN {X 0,Y 572.956,Z 518.909,A -85,B 0,C 180,E1 -2112.61,E2 -2112.61} C_VEL
LIN {X 0,Y 572.924,Z 518.858,A -85,B 0,C 180,E1 -2113.635,E2 -2113.635} C_VEL
LIN {X 0,Y 572.965,Z 517.961,A -85,B 0,C 180,E1 -2114.649,E2 -2114.649} C_VEL
LIN {X 0,Y 572.973,Z 516.264,A -85,B 0,C 180,E1 -2115.641,E2 -2115.641} C_VEL
LIN {X 0,Y 572.958,Z 513.798,A -85,B 0,C 180,E1 -2116.614,E2 -2116.614} C_VEL
LIN {X 0,Y 573.012,Z 510.529,A -85,B 0,C 180,E1 -2117.579,E2 -2117.579} C_VEL
LIN {X 0,Y 573.042,Z 505.246,A -85,B 0,C 180,E1 -2118.76,E2 -2118.76} C_VEL
LIN {X 0,Y 573.106,Z 498.421,A -85,B 0,C 180,E1 -2119.943,E2 -2119.943} C_VEL
LIN {X 0,Y 573.157,Z 491.25,A -85,B 0,C 180,E1 -2120.938,E2 -2120.938} C_VEL
LIN {X 0,Y 573.243,Z 482.274,A -85,B 0,C 180,E1 -2121.944,E2 -2121.944} C_VEL
LIN {X 0,Y 573.346,Z 472.67,A -85,B 0,C 180,E1 -2122.821,E2 -2122.821} C_VEL
LIN {X 0,Y 573.489,Z 461.512,A -85,B 0,C 180,E1 -2123.642,E2 -2123.642} C_VEL
LIN {X 0,Y 573.593,Z 449.093,A -85,B 0,C 180,E1 -2124.355,E2 -2124.355} C_VEL
LIN {X 0,Y 573.715,Z 437.935,A -85,B 0,C 180,E1 -2124.848,E2 -2124.848} C_VEL
LIN {X 0,Y 573.805,Z 424.907,A -85,B 0,C 180,E1 -2125.269,E2 -2125.269} C_VEL
LIN {X 0,Y 573.614,Z 418.873,A -85,B 0,C 180,E1 -2125.416,E2 -2125.416} C_VEL
LIN {X 0,Y 572.978,Z 414.903,A -85,B 0,C 180,E1 -2125.523,E2 -2125.523} C_VEL
LIN {X 0,Y 572.972,Z 410.363,A -85,B 0,C 180,E1 -2128.168,E2 -2128.168} C_VEL
LIN {X 0,Y 572.992,Z 406.206,A -85,B 0,C 180,E1 -2130.619,E2 -2130.619} C_VEL
LIN {X 0,Y 573.018,Z 401.306,A -85,B 0,C 180,E1 -2133.55,E2 -2133.55} C_VEL
LIN {X 0,Y 573.03,Z 397.079,A -85,B 0,C 180,E1 -2136.126,E2 -2136.126} C_VEL
LIN {X 0,Y 573.1,Z 392.446,A -85,B 0,C 180,E1 -2139.168,E2 -2139.168} C_VEL
LIN {X 0,Y 573.125,Z 389.161,A -85,B 0,C 180,E1 -2141.408,E2 -2141.408} C_VEL
LIN {X 0,Y 573.143,Z 385.724,A -85,B 0,C 180,E1 -2143.619,E2 -2143.619} C_VEL
LIN {X 0,Y 573.16,Z 381.32,A -85,B 0,C 180,E1 -2146.528,E2 -2146.528} C_VEL
LIN {X 0,Y 573.178,Z 379.19,A -85,B 0,C 180,E1 -2147.969,E2 -2147.969} C_VEL
LIN {X 0,Y 573.228,Z 379.085,A -85,B 0,C 180,E1 -2150.117,E2 -2150.117} C_VEL
LIN {X 0,Y 573.28,Z 379.079,A -85,B 0,C 180,E1 -2152.25,E2 -2152.25} C_VEL
LIN {X 0,Y 573.31,Z 379.073,A -85,B 0,C 180,E1 -2155.077,E2 -2155.077} C_VEL
LIN {X 0,Y 573.302,Z 379.075,A -85,B 0,C 180,E1 -2157.892,E2 -2157.892} C_VEL
LIN {X 0,Y 573.334,Z 379.072,A -85,B 0,C 180,E1 -2160.702,E2 -2160.702} C_VEL
LIN {X 0,Y 573.235,Z 379.083,A -85,B 0,C 180,E1 -2163.515,E2 -2163.515} C_VEL
LIN {X 0,Y 573.29,Z 379.076,A -85,B 0,C 180,E1 -2165.628,E2 -2165.628} C_VEL
LIN {X 0,Y 573.287,Z 379.076,A -85,B 0,C 180,E1 -2168.46,E2 -2168.46} C_VEL
LIN {X 0,Y 573.267,Z 379.079,A -85,B 0,C 180,E1 -2171.312,E2 -2171.312} C_VEL
LIN {X 0,Y 573.27,Z 379.08,A -85,B 0,C 180,E1 -2174.193,E2 -2174.193} C_VEL
LIN {X 0,Y 573.258,Z 379.08,A -85,B 0,C 180,E1 -2177.112,E2 -2177.112} C_VEL
LIN {X 0,Y 573.254,Z 379.08,A -85,B 0,C 180,E1 -2180.077,E2 -2180.077} C_VEL
LIN {X 0,Y 573.235,Z 379.083,A -85,B 0,C 180,E1 -2182.338,E2 -2182.338} C_VEL
LIN {X 0,Y 573.253,Z 379.081,A -85,B 0,C 180,E1 -2185.41,E2 -2185.41} C_VEL
LIN {X 0,Y 573.261,Z 379.08,A -85,B 0,C 180,E1 -2188.032,E2 -2188.032} C_VEL
LIN {X 0,Y 573.236,Z 379.085,A -85,B 0,C 180,E1 -2190.885,E2 -2190.885} C_VEL
LIN {X 0,Y 573.259,Z 379.079,A -85,B 0,C 180,E1 -2193.524,E2 -2193.524} C_VEL
LIN {X 0,Y 573.255,Z 379.082,A -85,B 0,C 180,E1 -2196.049,E2 -2196.049} C_VEL
LIN {X 0,Y 573.248,Z 379.081,A -85,B 0,C 180,E1 -2198.701,E2 -2198.701} C_VEL
LIN {X 0,Y 573.252,Z 379.081,A -85,B 0,C 180,E1 -2201.596,E2 -2201.596} C_VEL
LIN {X 0,Y 573.233,Z 379.085,A -85,B 0,C 180,E1 -2204.334,E2 -2204.334} C_VEL
LIN {X 0,Y 573.239,Z 379.083,A -85,B 0,C 180,E1 -2207.359,E2 -2207.359} C_VEL
LIN {X 0,Y 573.246,Z 379.082,A -85,B 0,C 180,E1 -2210.394,E2 -2210.394} C_VEL
LIN {X 0,Y 573.31,Z 379.135,A -85,B 0,C 180,E1 -2213.521,E2 -2213.521} C_VEL
LIN {X 0,Y 573.609,Z 383.462,A -85,B 0,C 180,E1 -2215.175,E2 -2215.175} C_VEL
LIN {X 0,Y 573.499,Z 390.549,A -85,B 0,C 180,E1 -2217.733,E2 -2217.733} C_VEL
LIN {X 0,Y 573.459,Z 399.109,A -85,B 0,C 180,E1 -2220.646,E2 -2220.646} C_VEL
LIN {X 0,Y 573.342,Z 408.718,A -85,B 0,C 180,E1 -2223.815,E2 -2223.815} C_VEL
LIN {X 0,Y 573.271,Z 417.063,A -85,B 0,C 180,E1 -2226.521,E2 -2226.521} C_VEL
LIN {X 0,Y 573.233,Z 425.345,A -85,B 0,C 180,E1 -2229.173,E2 -2229.173} C_VEL
LIN {X 0,Y 573.151,Z 434.811,A -85,B 0,C 180,E1 -2232.149,E2 -2232.149} C_VEL
LIN {X 0,Y 573.105,Z 443.095,A -85,B 0,C 180,E1 -2234.713,E2 -2234.713} C_VEL
LIN {X 0,Y 573.079,Z 452.192,A -85,B 0,C 180,E1 -2237.495,E2 -2237.495} C_VEL
LIN {X 0,Y 573.867,Z 458.388,A -85,B 0,C 180,E1 -2237.625,E2 -2237.625} C_VEL
LIN {X 0,Y 573.782,Z 470.511,A -85,B 0,C 180,E1 -2237.937,E2 -2237.937} C_VEL
LIN {X 0,Y 573.634,Z 483.469,A -85,B 0,C 180,E1 -2238.425,E2 -2238.425} C_VEL
LIN {X 0,Y 573.528,Z 496.03,A -85,B 0,C 180,E1 -2239.065,E2 -2239.065} C_VEL
LIN {X 0,Y 573.456,Z 506.751,A -85,B 0,C 180,E1 -2239.764,E2 -2239.764} C_VEL
LIN {X 0,Y 573.308,Z 515.651,A -85,B 0,C 180,E1 -2240.475,E2 -2240.475} C_VEL
LIN {X 0,Y 573.215,Z 524.79,A -85,B 0,C 180,E1 -2241.362,E2 -2241.362} C_VEL
LIN {X 0,Y 573.142,Z 533.692,A -85,B 0,C 180,E1 -2242.426,E2 -2242.426} C_VEL
LIN {X 0,Y 573.043,Z 540.45,A -85,B 0,C 180,E1 -2243.422,E2 -2243.422} C_VEL
LIN {X 0,Y 573.07,Z 545.682,A -85,B 0,C 180,E1 -2244.37,E2 -2244.37} C_VEL
LIN {X 0,Y 573.028,Z 550.373,A -85,B 0,C 180,E1 -2245.428,E2 -2245.428} C_VEL
LIN {X 0,Y 573.022,Z 553.958,A -85,B 0,C 180,E1 -2246.484,E2 -2246.484} C_VEL
LIN {X 0,Y 572.959,Z 555.809,A -85,B 0,C 180,E1 -2247.188,E2 -2247.188} C_VEL
LIN {X 0,Y 572.939,Z 557.199,A -85,B 0,C 180,E1 -2247.891,E2 -2247.891} C_VEL
LIN {X 0,Y 572.94,Z 558.785,A -85,B 0,C 180,E1 -2249.297,E2 -2249.297} C_VEL
LIN {X 0,Y 572.938,Z 559,A -85,B 0,C 180,E1 -2250,E2 -2250} C_VEL
LIN {X 0,Y 572.946,Z 558.186,A -85,B 0,C 180,E1 -2251.406,E2 -2251.406} C_VEL
LIN {X 0,Y 572.939,Z 557.2,A -85,B 0,C 180,E1 -2252.109,E2 -2252.109} C_VEL
LIN {X 0,Y 572.959,Z 555.809,A -85,B 0,C 180,E1 -2252.813,E2 -2252.813} C_VEL
LIN {X 0,Y 573.015,Z 552.895,A -85,B 0,C 180,E1 -2253.868,E2 -2253.868} C_VEL
LIN {X 0,Y 572.963,Z 548.948,A -85,B 0,C 180,E1 -2254.926,E2 -2254.926} C_VEL
LIN {X 0,Y 573.064,Z 542.876,A -85,B 0,C 180,E1 -2256.16,E2 -2256.16} C_VEL
LIN {X 0,Y 573.119,Z 536.236,A -85,B 0,C 180,E1 -2257.221,E2 -2257.221} C_VEL
LIN {X 0,Y 573.201,Z 527.989,A -85,B 0,C 180,E1 -2258.283,E2 -2258.283} C_VEL
LIN {X 0,Y 573.287,Z 519.536,A -85,B 0,C 180,E1 -2259.17,E2 -2259.17} C_VEL
LIN {X 0,Y 573.417,Z 509.095,A -85,B 0,C 180,E1 -2260.059,E2 -2260.059} C_VEL
LIN {X 0,Y 573.523,Z 497.524,A -85,B 0,C 180,E1 -2260.848,E2 -2260.848} C_VEL
LIN {X 0,Y 573.61,Z 485.878,A -85,B 0,C 180,E1 -2261.466,E2 -2261.466} C_VEL
LIN {X 0,Y 573.76,Z 473.168,A -85,B 0,C 180,E1 -2261.974,E2 -2261.974} C_VEL
LIN {X 0,Y 573.863,Z 460.512,A -85,B 0,C 180,E1 -2262.331,E2 -2262.331} C_VEL
LIN {X 0,Y 573.55,Z 455.222,A -85,B 0,C 180,E1 -2262.444,E2 -2262.444} C_VEL
LIN {X 0,Y 573.079,Z 452.19,A -85,B 0,C 180,E1 -2262.505,E2 -2262.505} C_VEL
LIN {X 0,Y 573.105,Z 443.093,A -85,B 0,C 180,E1 -2265.287,E2 -2265.287} C_VEL
LIN {X 0,Y 573.152,Z 434.81,A -85,B 0,C 180,E1 -2267.852,E2 -2267.852} C_VEL
LIN {X 0,Y 573.234,Z 425.343,A -85,B 0,C 180,E1 -2270.827,E2 -2270.827} C_VEL
LIN {X 0,Y 573.272,Z 417.061,A -85,B 0,C 180,E1 -2273.48,E2 -2273.48} C_VEL
LIN {X 0,Y 573.341,Z 407.714,A -85,B 0,C 180,E1 -2276.513,E2 -2276.513} C_VEL
LIN {X 0,Y 573.455,Z 398.599,A -85,B 0,C 180,E1 -2279.524,E2 -2279.524} C_VEL
LIN {X 0,Y 573.562,Z 389.609,A -85,B 0,C 180,E1 -2282.625,E2 -2282.625} C_VEL
LIN {X 0,Y 573.613,Z 382.619,A -85,B 0,C 180,E1 -2285.159,E2 -2285.159} C_VEL
LIN {X 0,Y 573.236,Z 379.085,A -85,B 0,C 180,E1 -2286.54,E2 -2286.54} C_VEL
LIN {X 0,Y 573.248,Z 379.081,A -85,B 0,C 180,E1 -2289.607,E2 -2289.607} C_VEL
LIN {X 0,Y 573.241,Z 379.082,A -85,B 0,C 180,E1 -2292.641,E2 -2292.641} C_VEL
LIN {X 0,Y 573.235,Z 379.083,A -85,B 0,C 180,E1 -2295.666,E2 -2295.666} C_VEL
LIN {X 0,Y 573.229,Z 379.083,A -85,B 0,C 180,E1 -2298.543,E2 -2298.543} C_VEL
LIN {X 0,Y 573.243,Z 379.08,A -85,B 0,C 180,E1 -2301.298,E2 -2301.298} C_VEL
LIN {X 0,Y 573.244,Z 379.082,A -85,B 0,C 180,E1 -2304.014,E2 -2304.014} C_VEL
LIN {X 0,Y 573.24,Z 379.083,A -85,B 0,C 180,E1 -2306.516,E2 -2306.516} C_VEL
LIN {X 0,Y 573.23,Z 379.085,A -85,B 0,C 180,E1 -2309.118,E2 -2309.118} C_VEL
LIN {X 0,Y 573.239,Z 379.084,A -85,B 0,C 180,E1 -2311.435,E2 -2311.435} C_VEL
LIN {X 0,Y 573.262,Z 379.081,A -85,B 0,C 180,E1 -2313.81,E2 -2313.81} C_VEL
LIN {X 0,Y 573.233,Z 379.084,A -85,B 0,C 180,E1 -2316.134,E2 -2316.134} C_VEL
LIN {X 0,Y 573.252,Z 379.079,A -85,B 0,C 180,E1 -2319.174,E2 -2319.174} C_VEL
LIN {X 0,Y 573.222,Z 379.083,A -85,B 0,C 180,E1 -2321.411,E2 -2321.411} C_VEL
LIN {X 0,Y 573.248,Z 379.08,A -85,B 0,C 180,E1 -2323.622,E2 -2323.622} C_VEL
LIN {X 0,Y 573.273,Z 379.079,A -85,B 0,C 180,E1 -2325.807,E2 -2325.807} C_VEL
